LIN {X 70.467,Y 80.092,Z 59.000,A 180.000,B 0.000,C 180.000} C_DIS
LIN {X 70.403,Y 79.913,Z 59.000,A 180.000,B 0.000,C 180.000} C_DIS
LIN {X 70.344,Y 79.735,Z 59.000,A 180.000,B 0.000,C 180.000} C_DIS
LIN {X 70.240,Y 79.377,Z 59.000,A 180.000,B 0.000,C 180.000} C_DIS
LIN {X 70.200,Y 79.198,Z 59.000,A 180.000,B 0.000,C 180.000} C_DIS
LIN {X 70.160,Y 79.020,Z 59.000,A 180.000,B 0.000,C 180.000} C_DIS
LIN {X 70.124,Y 78.841,Z 59.000,A 180.000,B 0.000,C 180.000} C_DIS
LIN {X 70.067,Y 78.483,Z 59.000,A 180.000,B 0.000,C 180.000} C_DIS
LIN {X 70.048,Y 78.304,Z 59.000,A 180.000,B 0.000,C 180.000} C_DIS
LIN {X 70.031,Y 78.126,Z 59.000,A 180.000,B 0.000,C 180.000} C_DIS
LIN {X 70.015,Y 77.947,Z 59.000,A 180.000,B 0.000,C 180.000} C_DIS
LIN {X 70.004,Y 77.589,Z 59.000,A 180.000,B 0.000,C 180.000} C_DIS
LIN {X 70.004,Y 77.411,Z 59.000,A 180.000,B 0.000,C 180.000} C_DIS
LIN {X 70.015,Y 77.053,Z 59.000,A 180.000,B 0.000,C 180.000} C_DIS
LIN {X 70.031,Y 76.874,Z 59.000,A 180.000,B 0.000,C 180.000} C_DIS
LIN {X 70.048,Y 76.696,Z 59.000,A 180.000,B 0.000,C 180.000} C_DIS
LIN {X 70.067,Y 76.517,Z 59.000,A 180.000,B 0.000,C 180.000} C_DIS
LIN {X 70.124,Y 76.159,Z 59.000,A 180.000,B 0.000,C 180.000} C_DIS
LIN {X 70.160,Y 75.980,Z 59.000,A 180.000,B 0.000,C 180.000} C_DIS
LIN {X 70.200,Y 75.802,Z 59.000,A 180.000,B 0.000,C 180.000} C_DIS
LIN {X 70.240,Y 75.623,Z 59.000,A 180.000,B 0.000,C 180.000} C_DIS
LIN {X 70.344,Y 75.265,Z 59.000,A 180.000,B 0.000,C 180.000} C_DIS
LIN {X 70.403,Y 75.087,Z 59.000,A 180.000,B 0.000,C 180.000} C_DIS
LIN {X 70.467,Y 74.908,Z 59.000,A 180.000,B 0.000,C 180.000} C_DIS
LIN {X 70.501,Y 74.814,Z 59.000,A 180.000,B 0.000,C 180.000} C_DIS
LIN {X 70.532,Y 74.729,Z 59.000,A 180.000,B 0.000,C 180.000} C_DIS
LIN {X 70.687,Y 74.372,Z 59.000,A 180.000,B 0.000,C 180.000} C_DIS
LIN {X 70.773,Y 74.193,Z 59.000,A 180.000,B 0.000,C 180.000} C_DIS
LIN {X 70.864,Y 74.014,Z 59.000,A 180.000,B 0.000,C 180.000} C_DIS
LIN {X 70.960,Y 73.835,Z 59.000,A 180.000,B 0.000,C 180.000} C_DIS
LIN {X 71.154,Y 73.507,Z 59.000,A 180.000,B 0.000,C 180.000} C_DIS
LIN {X 71.171,Y 73.478,Z 59.000,A 180.000,B 0.000,C 180.000} C_DIS
LIN {X 71.414,Y 73.120,Z 59.000,A 180.000,B 0.000,C 180.000} C_DIS
LIN {X 71.511,Y 72.992,Z 59.000,A 180.000,B 0.000,C 180.000} C_DIS
LIN {X 71.690,Y 72.762,Z 59.000,A 180.000,B 0.000,C 180.000} C_DIS
LIN {X 71.842,Y 72.584,Z 59.000,A 180.000,B 0.000,C 180.000} C_DIS
LIN {X 72.000,Y 72.405,Z 59.000,A 180.000,B 0.000,C 180.000} C_DIS
LIN {X 72.048,Y 72.353,Z 59.000,A 180.000,B 0.000,C 180.000} C_DIS
LIN {X 72.353,Y 72.048,Z 59.000,A 180.000,B 0.000,C 180.000} C_DIS
LIN {X 72.405,Y 72.000,Z 59.000,A 180.000,B 0.000,C 180.000} C_DIS
LIN {X 72.584,Y 71.842,Z 59.000,A 180.000,B 0.000,C 180.000} C_DIS
LIN {X 72.762,Y 71.690,Z 59.000,A 180.000,B 0.000,C 180.000} C_DIS
LIN {X 72.992,Y 71.511,Z 59.000,A 180.000,B 0.000,C 180.000} C_DIS
LIN {X 73.120,Y 71.414,Z 59.000,A 180.000,B 0.000,C 180.000} C_DIS
LIN {X 73.478,Y 71.171,Z 59.000,A 180.000,B 0.000,C 180.000} C_DIS
LIN {X 73.507,Y 71.154,Z 59.000,A 180.000,B 0.000,C 180.000} C_DIS
LIN {X 73.835,Y 70.960,Z 59.000,A 180.000,B 0.000,C 180.000} C_DIS
LIN {X 74.014,Y 70.864,Z 59.000,A 180.000,B 0.000,C 180.000} C_DIS
LIN {X 74.193,Y 70.773,Z 59.000,A 180.000,B 0.000,C 180.000} C_DIS
LIN {X 74.372,Y 70.687,Z 59.000,A 180.000,B 0.000,C 180.000} C_DIS
LIN {X 74.729,Y 70.532,Z 59.000,A 180.000,B 0.000,C 180.000} C_DIS
LIN {X 74.908,Y 70.467,Z 59.000,A 180.000,B 0.000,C 180.000} C_DIS
LIN {X 75.087,Y 70.403,Z 59.000,A 180.000,B 0.000,C 180.000} C_DIS
LIN {X 75.265,Y 70.344,Z 59.000,A 180.000,B 0.000,C 180.000} C_DIS
LIN {X 75.623,Y 70.240,Z 59.000,A 180.000,B 0.000,C 180.000} C_DIS
LIN {X 75.802,Y 70.200,Z 59.000,A 180.000,B 0.000,C 180.000} C_DIS
LIN {X 75.980,Y 70.160,Z 59.000,A 180.000,B 0.000,C 180.000} C_DIS
LIN {X 76.159,Y 70.124,Z 59.000,A 180.000,B 0.000,C 180.000} C_DIS
LIN {X 76.517,Y 70.067,Z 59.000,A 180.000,B 0.000,C 180.000} C_DIS
LIN {X 76.696,Y 70.048,Z 59.000,A 180.000,B 0.000,C 180.000} C_DIS
LIN {X 76.874,Y 70.031,Z 59.000,A 180.000,B 0.000,C 180.000} C_DIS
LIN {X 77.053,Y 70.015,Z 59.000,A 180.000,B 0.000,C 180.000} C_DIS
LIN {X 77.411,Y 70.004,Z 59.000,A 180.000,B 0.000,C 180.000} C_DIS
LIN {X 77.589,Y 70.004,Z 59.000,A 180.000,B 0.000,C 180.000} C_DIS
LIN {X 77.947,Y 70.015,Z 59.000,A 180.000,B 0.000,C 180.000} C_DIS
LIN {X 78.126,Y 70.031,Z 59.000,A 180.000,B 0.000,C 180.000} C_DIS
LIN {X 78.304,Y 70.048,Z 59.000,A 180.000,B 0.000,C 180.000} C_DIS
LIN {X 78.483,Y 70.067,Z 59.000,A 180.000,B 0.000,C 180.000} C_DIS
LIN {X 78.841,Y 70.124,Z 59.000,A 180.000,B 0.000,C 180.000} C_DIS
LIN {X 79.020,Y 70.160,Z 59.000,A 180.000,B 0.000,C 180.000} C_DIS
LIN {X 79.198,Y 70.200,Z 59.000,A 180.000,B 0.000,C 180.000} C_DIS
LIN {X 79.377,Y 70.240,Z 59.000,A 180.000,B 0.000,C 180.000} C_DIS
LIN {X 79.735,Y 70.344,Z 59.000,A 180.000,B 0.000,C 180.000} C_DIS
LIN {X 79.913,Y 70.403,Z 59.000,A 180.000,B 0.000,C 180.000} C_DIS
LIN {X 80.092,Y 70.467,Z 59.000,A 180.000,B 0.000,C 180.000} C_DIS
LIN {X 80.271,Y 70.532,Z 59.000,A 180.000,B 0.000,C 180.000} C_DIS
LIN {X 80.628,Y 70.687,Z 59.000,A 180.000,B 0.000,C 180.000} C_DIS
LIN {X 80.807,Y 70.773,Z 59.000,A 180.000,B 0.000,C 180.000} C_DIS
LIN {X 80.986,Y 70.864,Z 59.000,A 180.000,B 0.000,C 180.000} C_DIS
LIN {X 81.165,Y 70.960,Z 59.000,A 180.000,B 0.000,C 180.000} C_DIS
LIN {X 81.493,Y 71.154,Z 59.000,A 180.000,B 0.000,C 180.000} C_DIS
LIN {X 81.522,Y 71.171,Z 59.000,A 180.000,B 0.000,C 180.000} C_DIS
LIN {X 81.880,Y 71.414,Z 59.000,A 180.000,B 0.000,C 180.000} C_DIS
LIN {X 82.008,Y 71.511,Z 59.000,A 180.000,B 0.000,C 180.000} C_DIS
LIN {X 82.238,Y 71.690,Z 59.000,A 180.000,B 0.000,C 180.000} C_DIS
LIN {X 82.416,Y 71.842,Z 59.000,A 180.000,B 0.000,C 180.000} C_DIS
LIN {X 82.595,Y 72.000,Z 59.000,A 180.000,B 0.000,C 180.000} C_DIS
LIN {X 82.647,Y 72.048,Z 59.000,A 180.000,B 0.000,C 180.000} C_DIS
LIN {X 82.952,Y 72.353,Z 59.000,A 180.000,B 0.000,C 180.000} C_DIS
LIN {X 83.000,Y 72.405,Z 59.000,A 180.000,B 0.000,C 180.000} C_DIS
LIN {X 83.158,Y 72.584,Z 59.000,A 180.000,B 0.000,C 180.000} C_DIS
LIN {X 83.310,Y 72.762,Z 59.000,A 180.000,B 0.000,C 180.000} C_DIS
LIN {X 83.489,Y 72.992,Z 59.000,A 180.000,B 0.000,C 180.000} C_DIS
LIN {X 83.586,Y 73.120,Z 59.000,A 180.000,B 0.000,C 180.000} C_DIS
LIN {X 83.829,Y 73.478,Z 59.000,A 180.000,B 0.000,C 180.000} C_DIS
LIN {X 83.846,Y 73.507,Z 59.000,A 180.000,B 0.000,C 180.000} C_DIS
LIN {X 84.040,Y 73.835,Z 59.000,A 180.000,B 0.000,C 180.000} C_DIS
LIN {X 84.136,Y 74.014,Z 59.000,A 180.000,B 0.000,C 180.000} C_DIS
LIN {X 84.227,Y 74.193,Z 59.000,A 180.000,B 0.000,C 180.000} C_DIS
LIN {X 84.313,Y 74.372,Z 59.000,A 180.000,B 0.000,C 180.000} C_DIS
LIN {X 84.468,Y 74.729,Z 59.000,A 180.000,B 0.000,C 180.000} C_DIS
LIN {X 84.533,Y 74.908,Z 59.000,A 180.000,B 0.000,C 180.000} C_DIS
LIN {X 84.597,Y 75.087,Z 59.000,A 180.000,B 0.000,C 180.000} C_DIS
LIN {X 84.656,Y 75.265,Z 59.000,A 180.000,B 0.000,C 180.000} C_DIS
LIN {X 84.760,Y 75.623,Z 59.000,A 180.000,B 0.000,C 180.000} C_DIS
LIN {X 84.800,Y 75.802,Z 59.000,A 180.000,B 0.000,C 180.000} C_DIS
LIN {X 84.840,Y 75.980,Z 59.000,A 180.000,B 0.000,C 180.000} C_DIS
LIN {X 84.876,Y 76.159,Z 59.000,A 180.000,B 0.000,C 180.000} C_DIS
LIN {X 84.933,Y 76.517,Z 59.000,A 180.000,B 0.000,C 180.000} C_DIS
LIN {X 84.952,Y 76.696,Z 59.000,A 180.000,B 0.000,C 180.000} C_DIS
LIN {X 84.969,Y 76.874,Z 59.000,A 180.000,B 0.000,C 180.000} C_DIS
LIN {X 84.985,Y 77.053,Z 59.000,A 180.000,B 0.000,C 180.000} C_DIS
LIN {X 84.996,Y 77.411,Z 59.000,A 180.000,B 0.000,C 180.000} C_DIS
LIN {X 84.996,Y 77.589,Z 59.000,A 180.000,B 0.000,C 180.000} C_DIS
LIN {X 84.985,Y 77.947,Z 59.000,A 180.000,B 0.000,C 180.000} C_DIS
LIN {X 84.969,Y 78.126,Z 59.000,A 180.000,B 0.000,C 180.000} C_DIS
LIN {X 84.952,Y 78.304,Z 59.000,A 180.000,B 0.000,C 180.000} C_DIS
LIN {X 84.933,Y 78.483,Z 59.000,A 180.000,B 0.000,C 180.000} C_DIS
LIN {X 84.876,Y 78.841,Z 59.000,A 180.000,B 0.000,C 180.000} C_DIS
LIN {X 84.840,Y 79.020,Z 59.000,A 180.000,B 0.000,C 180.000} C_DIS
LIN {X 84.800,Y 79.198,Z 59.000,A 180.000,B 0.000,C 180.000} C_DIS
LIN {X 84.760,Y 79.377,Z 59.000,A 180.000,B 0.000,C 180.000} C_DIS
LIN {X 84.656,Y 79.735,Z 59.000,A 180.000,B 0.000,C 180.000} C_DIS
LIN {X 84.597,Y 79.913,Z 59.000,A 180.000,B 0.000,C 180.000} C_DIS
LIN {X 84.533,Y 80.092,Z 59.000,A 180.000,B 0.000,C 180.000} C_DIS
LIN {X 84.468,Y 80.271,Z 59.000,A 180.000,B 0.000,C 180.000} C_DIS
LIN {X 84.313,Y 80.628,Z 59.000,A 180.000,B 0.000,C 180.000} C_DIS
LIN {X 84.227,Y 80.807,Z 59.000,A 180.000,B 0.000,C 180.000} C_DIS
LIN {X 84.136,Y 80.986,Z 59.000,A 180.000,B 0.000,C 180.000} C_DIS
LIN {X 84.040,Y 81.165,Z 59.000,A 180.000,B 0.000,C 180.000} C_DIS
LIN {X 83.846,Y 81.493,Z 59.000,A 180.000,B 0.000,C 180.000} C_DIS
LIN {X 83.829,Y 81.522,Z 59.000,A 180.000,B 0.000,C 180.000} C_DIS
LIN {X 83.586,Y 81.880,Z 59.000,A 180.000,B 0.000,C 180.000} C_DIS
LIN {X 83.489,Y 82.008,Z 59.000,A 180.000,B 0.000,C 180.000} C_DIS
LIN {X 83.310,Y 82.238,Z 59.000,A 180.000,B 0.000,C 180.000} C_DIS
LIN {X 83.158,Y 82.416,Z 59.000,A 180.000,B 0.000,C 180.000} C_DIS
LIN {X 83.000,Y 82.595,Z 59.000,A 180.000,B 0.000,C 180.000} C_DIS
LIN {X 82.952,Y 82.647,Z 59.000,A 180.000,B 0.000,C 180.000} C_DIS
LIN {X 82.647,Y 82.952,Z 59.000,A 180.000,B 0.000,C 180.000} C_DIS
LIN {X 82.595,Y 83.000,Z 59.000,A 180.000,B 0.000,C 180.000} C_DIS
LIN {X 82.416,Y 83.158,Z 59.000,A 180.000,B 0.000,C 180.000} C_DIS
LIN {X 82.238,Y 83.310,Z 59.000,A 180.000,B 0.000,C 180.000} C_DIS
LIN {X 82.008,Y 83.489,Z 59.000,A 180.000,B 0.000,C 180.000} C_DIS
LIN {X 81.880,Y 83.586,Z 59.000,A 180.000,B 0.000,C 180.000} C_DIS
LIN {X 81.522,Y 83.829,Z 59.000,A 180.000,B 0.000,C 180.000} C_DIS
LIN {X 81.493,Y 83.846,Z 59.000,A 180.000,B 0.000,C 180.000} C_DIS
LIN {X 81.165,Y 84.040,Z 59.000,A 180.000,B 0.000,C 180.000} C_DIS
LIN {X 80.986,Y 84.136,Z 59.000,A 180.000,B 0.000,C 180.000} C_DIS
LIN {X 80.807,Y 84.227,Z 59.000,A 180.000,B 0.000,C 180.000} C_DIS
LIN {X 80.628,Y 84.313,Z 59.000,A 180.000,B 0.000,C 180.000} C_DIS
LIN {X 80.271,Y 84.468,Z 59.000,A 180.000,B 0.000,C 180.000} C_DIS
LIN {X 80.092,Y 84.533,Z 59.000,A 180.000,B 0.000,C 180.000} C_DIS
LIN {X 79.913,Y 84.597,Z 59.000,A 180.000,B 0.000,C 180.000} C_DIS
LIN {X 79.735,Y 84.656,Z 59.000,A 180.000,B 0.000,C 180.000} C_DIS
LIN {X 79.377,Y 84.760,Z 59.000,A 180.000,B 0.000,C 180.000} C_DIS
LIN {X 79.198,Y 84.800,Z 59.000,A 180.000,B 0.000,C 180.000} C_DIS
LIN {X 79.020,Y 84.840,Z 59.000,A 180.000,B 0.000,C 180.000} C_DIS
LIN {X 78.841,Y 84.876,Z 59.000,A 180.000,B 0.000,C 180.000} C_DIS
LIN {X 78.483,Y 84.933,Z 59.000,A 180.000,B 0.000,C 180.000} C_DIS
LIN {X 78.304,Y 84.952,Z 59.000,A 180.000,B 0.000,C 180.000} C_DIS
LIN {X 78.126,Y 84.969,Z 59.000,A 180.000,B 0.000,C 180.000} C_DIS
LIN {X 77.947,Y 84.985,Z 59.000,A 180.000,B 0.000,C 180.000} C_DIS
LIN {X 77.589,Y 84.996,Z 59.000,A 180.000,B 0.000,C 180.000} C_DIS
LIN {X 77.411,Y 84.996,Z 59.000,A 180.000,B 0.000,C 180.000} C_DIS
LIN {X 77.053,Y 84.985,Z 59.000,A 180.000,B 0.000,C 180.000} C_DIS
LIN {X 76.874,Y 84.969,Z 59.000,A 180.000,B 0.000,C 180.000} C_DIS
LIN {X 76.696,Y 84.952,Z 59.000,A 180.000,B 0.000,C 180.000} C_DIS
LIN {X 76.517,Y 84.933,Z 59.000,A 180.000,B 0.000,C 180.000} C_DIS
LIN {X 76.159,Y 84.876,Z 59.000,A 180.000,B 0.000,C 180.000} C_DIS
LIN {X 75.980,Y 84.840,Z 59.000,A 180.000,B 0.000,C 180.000} C_DIS
LIN {X 75.802,Y 84.800,Z 59.000,A 180.000,B 0.000,C 180.000} C_DIS
LIN {X 75.623,Y 84.760,Z 59.000,A 180.000,B 0.000,C 180.000} C_DIS
LIN {X 75.265,Y 84.656,Z 59.000,A 180.000,B 0.000,C 180.000} C_DIS
LIN {X 75.087,Y 84.597,Z 59.000,A 180.000,B 0.000,C 180.000} C_DIS
LIN {X 74.908,Y 84.533,Z 59.000,A 180.000,B 0.000,C 180.000} C_DIS
LIN {X 74.729,Y 84.468,Z 59.000,A 180.000,B 0.000,C 180.000} C_DIS
LIN {X 74.372,Y 84.313,Z 59.000,A 180.000,B 0.000,C 180.000} C_DIS
LIN {X 74.193,Y 84.227,Z 59.000,A 180.000,B 0.000,C 180.000} C_DIS
LIN {X 74.014,Y 84.136,Z 59.000,A 180.000,B 0.000,C 180.000} C_DIS
LIN {X 73.835,Y 84.040,Z 59.000,A 180.000,B 0.000,C 180.000} C_DIS
LIN {X 73.507,Y 83.846,Z 59.000,A 180.000,B 0.000,C 180.000} C_DIS
LIN {X 73.478,Y 83.829,Z 59.000,A 180.000,B 0.000,C 180.000} C_DIS
LIN {X 73.260,Y 83.681,Z 59.000,A 180.000,B 0.000,C 180.000} C_DIS
; Link Move Starts
LIN {X 73.004,Y 83.498,Z 59.000,A 180.000,B 0.000,C 180.000} C_DIS
LIN {X 72.755,Y 83.305,Z 58.999,A 180.000,B 0.000,C 180.000} C_DIS
LIN {X 72.517,Y 83.099,Z 58.998,A 180.000,B 0.000,C 180.000} C_DIS
LIN {X 72.286,Y 82.885,Z 58.996,A 180.000,B 0.000,C 180.000} C_DIS
LIN {X 72.063,Y 82.663,Z 58.994,A 180.000,B 0.000,C 180.000} C_DIS
LIN {X 71.853,Y 82.428,Z 58.991,A 180.000,B 0.000,C 180.000} C_DIS
LIN {X 71.650,Y 82.187,Z 58.988,A 180.000,B 0.000,C 180.000} C_DIS
LIN {X 71.457,Y 81.938,Z 58.985,A 180.000,B 0.000,C 180.000} C_DIS
LIN {X 71.278,Y 81.679,Z 58.981,A 180.000,B 0.000,C 180.000} C_DIS
LIN {X 71.107,Y 81.414,Z 58.977,A 180.000,B 0.000,C 180.000} C_DIS
LIN {X 70.947,Y 81.143,Z 58.972,A 180.000,B 0.000,C 180.000} C_DIS
LIN {X 70.873,Y 81.004,Z 58.969,A 180.000,B 0.000,C 180.000} C_DIS
LIN {X 70.802,Y 80.864,Z 58.967,A 180.000,B 0.000,C 180.000} C_DIS
LIN {X 70.730,Y 80.723,Z 58.964,A 180.000,B 0.000,C 180.000} C_DIS
LIN {X 70.666,Y 80.579,Z 58.961,A 180.000,B 0.000,C 180.000} C_DIS
LIN {X 70.603,Y 80.435,Z 58.959,A 180.000,B 0.000,C 180.000} C_DIS
LIN {X 70.541,Y 80.290,Z 58.956,A 180.000,B 0.000,C 180.000} C_DIS
LIN {X 70.485,Y 80.143,Z 58.952,A 180.000,B 0.000,C 180.000} C_DIS
LIN {X 70.432,Y 79.995,Z 58.949,A 180.000,B 0.000,C 180.000} C_DIS
LIN {X 70.379,Y 79.847,Z 58.946,A 180.000,B 0.000,C 180.000} C_DIS
LIN {X 70.333,Y 79.696,Z 58.943,A 180.000,B 0.000,C 180.000} C_DIS
LIN {X 70.289,Y 79.545,Z 58.939,A 180.000,B 0.000,C 180.000} C_DIS
LIN {X 70.245,Y 79.393,Z 58.936,A 180.000,B 0.000,C 180.000} C_DIS
LIN {X 70.209,Y 79.240,Z 58.932,A 180.000,B 0.000,C 180.000} C_DIS
LIN {X 70.175,Y 79.086,Z 58.928,A 180.000,B 0.000,C 180.000} C_DIS
LIN {X 70.140,Y 78.933,Z 58.925,A 180.000,B 0.000,C 180.000} C_DIS
LIN {X 70.114,Y 78.777,Z 58.921,A 180.000,B 0.000,C 180.000} C_DIS
LIN {X 70.089,Y 78.622,Z 58.917,A 180.000,B 0.000,C 180.000} C_DIS
LIN {X 70.065,Y 78.466,Z 58.913,A 180.000,B 0.000,C 180.000} C_DIS
LIN {X 70.048,Y 78.310,Z 58.909,A 180.000,B 0.000,C 180.000} C_DIS
LIN {X 70.033,Y 78.153,Z 58.905,A 180.000,B 0.000,C 180.000} C_DIS
LIN {X 70.018,Y 77.996,Z 58.900,A 180.000,B 0.000,C 180.000} C_DIS
LIN {X 70.012,Y 77.839,Z 58.896,A 180.000,B 0.000,C 180.000} C_DIS
LIN {X 70.007,Y 77.681,Z 58.892,A 180.000,B 0.000,C 180.000} C_DIS
LIN {X 70.002,Y 77.524,Z 58.887,A 180.000,B 0.000,C 180.000} C_DIS
LIN {X 70.005,Y 77.366,Z 58.883,A 180.000,B 0.000,C 180.000} C_DIS
LIN {X 70.010,Y 77.209,Z 58.878,A 180.000,B 0.000,C 180.000} C_DIS
LIN {X 70.015,Y 77.051,Z 58.873,A 180.000,B 0.000,C 180.000} C_DIS
LIN {X 70.029,Y 76.894,Z 58.869,A 180.000,B 0.000,C 180.000} C_DIS
LIN {X 70.044,Y 76.738,Z 58.864,A 180.000,B 0.000,C 180.000} C_DIS
LIN {X 70.058,Y 76.581,Z 58.859,A 180.000,B 0.000,C 180.000} C_DIS
LIN {X 70.082,Y 76.425,Z 58.854,A 180.000,B 0.000,C 180.000} C_DIS
LIN {X 70.094,Y 76.347,Z 58.851,A 180.000,B 0.000,C 180.000} C_DIS
LIN {X 70.106,Y 76.270,Z 58.849,A 180.000,B 0.000,C 180.000} C_DIS
LIN {X 70.119,Y 76.192,Z 58.846,A 180.000,B 0.000,C 180.000} C_DIS
LIN {X 70.131,Y 76.114,Z 58.844,A 180.000,B 0.000,C 180.000} C_DIS
LIN {X 70.147,Y 76.037,Z 58.841,A 180.000,B 0.000,C 180.000} C_DIS
LIN {X 70.164,Y 75.960,Z 58.839,A 180.000,B 0.000,C 180.000} C_DIS
LIN {X 70.181,Y 75.883,Z 58.836,A 180.000,B 0.000,C 180.000} C_DIS
LIN {X 70.216,Y 75.729,Z 58.831,A 180.000,B 0.000,C 180.000} C_DIS
LIN {X 70.233,Y 75.653,Z 58.828,A 180.000,B 0.000,C 180.000} C_DIS
LIN {X 70.254,Y 75.577,Z 58.825,A 180.000,B 0.000,C 180.000} C_DIS
LIN {X 70.298,Y 75.425,Z 58.820,A 180.000,B 0.000,C 180.000} C_DIS
LIN {X 70.342,Y 75.274,Z 58.815,A 180.000,B 0.000,C 180.000} C_DIS
LIN {X 70.364,Y 75.198,Z 58.812,A 180.000,B 0.000,C 180.000} C_DIS
LIN {X 70.389,Y 75.124,Z 58.809,A 180.000,B 0.000,C 180.000} C_DIS
LIN {X 70.416,Y 75.050,Z 58.806,A 180.000,B 0.000,C 180.000} C_DIS
LIN {X 70.469,Y 74.902,Z 58.801,A 180.000,B 0.000,C 180.000} C_DIS
LIN {X 70.523,Y 74.754,Z 58.796,A 180.000,B 0.000,C 180.000} C_DIS
LIN {X 70.553,Y 74.681,Z 58.793,A 180.000,B 0.000,C 180.000} C_DIS
LIN {X 70.616,Y 74.536,Z 58.787,A 180.000,B 0.000,C 180.000} C_DIS
LIN {X 70.647,Y 74.464,Z 58.785,A 180.000,B 0.000,C 180.000} C_DIS
LIN {X 70.710,Y 74.320,Z 58.779,A 180.000,B 0.000,C 180.000} C_DIS
LIN {X 70.745,Y 74.249,Z 58.776,A 180.000,B 0.000,C 180.000} C_DIS
LIN {X 70.780,Y 74.179,Z 58.774,A 180.000,B 0.000,C 180.000} C_DIS
LIN {X 70.852,Y 74.038,Z 58.768,A 180.000,B 0.000,C 180.000} C_DIS
LIN {X 70.923,Y 73.898,Z 58.763,A 180.000,B 0.000,C 180.000} C_DIS
LIN {X 70.963,Y 73.830,Z 58.760,A 180.000,B 0.000,C 180.000} C_DIS
LIN {X 71.043,Y 73.694,Z 58.754,A 180.000,B 0.000,C 180.000} C_DIS
LIN {X 71.083,Y 73.627,Z 58.752,A 180.000,B 0.000,C 180.000} C_DIS
LIN {X 71.163,Y 73.491,Z 58.746,A 180.000,B 0.000,C 180.000} C_DIS
LIN {X 71.207,Y 73.425,Z 58.743,A 180.000,B 0.000,C 180.000} C_DIS
LIN {X 71.251,Y 73.360,Z 58.741,A 180.000,B 0.000,C 180.000} C_DIS
LIN {X 71.340,Y 73.230,Z 58.735,A 180.000,B 0.000,C 180.000} C_DIS
LIN {X 71.428,Y 73.100,Z 58.730,A 180.000,B 0.000,C 180.000} C_DIS
LIN {X 71.476,Y 73.037,Z 58.727,A 180.000,B 0.000,C 180.000} C_DIS
LIN {X 71.573,Y 72.913,Z 58.721,A 180.000,B 0.000,C 180.000} C_DIS
LIN {X 71.621,Y 72.851,Z 58.719,A 180.000,B 0.000,C 180.000} C_DIS
LIN {X 71.717,Y 72.726,Z 58.713,A 180.000,B 0.000,C 180.000} C_DIS
LIN {X 71.769,Y 72.667,Z 58.710,A 180.000,B 0.000,C 180.000} C_DIS
LIN {X 71.821,Y 72.608,Z 58.708,A 180.000,B 0.000,C 180.000} C_DIS
LIN {X 71.925,Y 72.489,Z 58.702,A 180.000,B 0.000,C 180.000} C_DIS
LIN {X 72.030,Y 72.371,Z 58.697,A 180.000,B 0.000,C 180.000} C_DIS
LIN {X 72.085,Y 72.315,Z 58.694,A 180.000,B 0.000,C 180.000} C_DIS
LIN {X 72.196,Y 72.204,Z 58.688,A 180.000,B 0.000,C 180.000} C_DIS
LIN {X 72.252,Y 72.148,Z 58.686,A 180.000,B 0.000,C 180.000} C_DIS
LIN {X 72.363,Y 72.037,Z 58.680,A 180.000,B 0.000,C 180.000} C_DIS
LIN {X 72.422,Y 71.985,Z 58.677,A 180.000,B 0.000,C 180.000} C_DIS
LIN {X 72.541,Y 71.880,Z 58.672,A 180.000,B 0.000,C 180.000} C_DIS
LIN {X 72.659,Y 71.776,Z 58.666,A 180.000,B 0.000,C 180.000} C_DIS
LIN {X 72.718,Y 71.724,Z 58.664,A 180.000,B 0.000,C 180.000} C_DIS
LIN {X 72.780,Y 71.676,Z 58.661,A 180.000,B 0.000,C 180.000} C_DIS
LIN {X 73.091,Y 71.434,Z 58.647,A 180.000,B 0.000,C 180.000} C_DIS
LIN {X 73.156,Y 71.390,Z 58.644,A 180.000,B 0.000,C 180.000} C_DIS
LIN {X 73.286,Y 71.301,Z 58.639,A 180.000,B 0.000,C 180.000} C_DIS
LIN {X 73.482,Y 71.169,Z 58.631,A 180.000,B 0.000,C 180.000} C_DIS
LIN {X 73.617,Y 71.089,Z 58.625,A 180.000,B 0.000,C 180.000} C_DIS
LIN {X 73.821,Y 70.968,Z 58.617,A 180.000,B 0.000,C 180.000} C_DIS
LIN {X 73.889,Y 70.928,Z 58.614,A 180.000,B 0.000,C 180.000} C_DIS
LIN {X 74.239,Y 70.749,Z 58.600,A 180.000,B 0.000,C 180.000} C_DIS
LIN {X 74.310,Y 70.714,Z 58.598,A 180.000,B 0.000,C 180.000} C_DIS
LIN {X 74.527,Y 70.620,Z 58.589,A 180.000,B 0.000,C 180.000} C_DIS
LIN {X 74.671,Y 70.557,Z 58.584,A 180.000,B 0.000,C 180.000} C_DIS
LIN {X 74.743,Y 70.526,Z 58.581,A 180.000,B 0.000,C 180.000} C_DIS
LIN {X 75.114,Y 70.393,Z 58.567,A 180.000,B 0.000,C 180.000} C_DIS
LIN {X 75.188,Y 70.367,Z 58.565,A 180.000,B 0.000,C 180.000} C_DIS
LIN {X 75.566,Y 70.257,Z 58.551,A 180.000,B 0.000,C 180.000} C_DIS
LIN {X 75.642,Y 70.235,Z 58.548,A 180.000,B 0.000,C 180.000} C_DIS
LIN {X 76.026,Y 70.149,Z 58.534,A 180.000,B 0.000,C 180.000} C_DIS
LIN {X 76.103,Y 70.133,Z 58.532,A 180.000,B 0.000,C 180.000} C_DIS
LIN {X 76.492,Y 70.071,Z 58.518,A 180.000,B 0.000,C 180.000} C_DIS
LIN {X 76.570,Y 70.059,Z 58.515,A 180.000,B 0.000,C 180.000} C_DIS
LIN {X 76.962,Y 70.022,Z 58.501,A 180.000,B 0.000,C 180.000} C_DIS
LIN {X 77.041,Y 70.016,Z 58.499,A 180.000,B 0.000,C 180.000} C_DIS
LIN {X 77.434,Y 70.003,Z 58.485,A 180.000,B 0.000,C 180.000} C_DIS
LIN {X 77.513,Y 70.002,Z 58.482,A 180.000,B 0.000,C 180.000} C_DIS
LIN {X 77.907,Y 70.014,Z 58.468,A 180.000,B 0.000,C 180.000} C_DIS
LIN {X 77.985,Y 70.017,Z 58.466,A 180.000,B 0.000,C 180.000} C_DIS
LIN {X 78.377,Y 70.054,Z 58.452,A 180.000,B 0.000,C 180.000} C_DIS
LIN {X 78.456,Y 70.063,Z 58.449,A 180.000,B 0.000,C 180.000} C_DIS
LIN {X 78.845,Y 70.124,Z 58.435,A 180.000,B 0.000,C 180.000} C_DIS
LIN {X 78.922,Y 70.138,Z 58.433,A 180.000,B 0.000,C 180.000} C_DIS
LIN {X 79.307,Y 70.224,Z 58.419,A 180.000,B 0.000,C 180.000} C_DIS
LIN {X 79.383,Y 70.242,Z 58.416,A 180.000,B 0.000,C 180.000} C_DIS
LIN {X 79.761,Y 70.352,Z 58.402,A 180.000,B 0.000,C 180.000} C_DIS
LIN {X 79.836,Y 70.375,Z 58.400,A 180.000,B 0.000,C 180.000} C_DIS
LIN {X 80.059,Y 70.455,Z 58.391,A 180.000,B 0.000,C 180.000} C_DIS
LIN {X 80.207,Y 70.509,Z 58.386,A 180.000,B 0.000,C 180.000} C_DIS
LIN {X 80.281,Y 70.537,Z 58.383,A 180.000,B 0.000,C 180.000} C_DIS
LIN {X 80.642,Y 70.693,Z 58.369,A 180.000,B 0.000,C 180.000} C_DIS
LIN {X 80.714,Y 70.726,Z 58.367,A 180.000,B 0.000,C 180.000} C_DIS
LIN {X 80.924,Y 70.833,Z 58.358,A 180.000,B 0.000,C 180.000} C_DIS
LIN {X 81.065,Y 70.904,Z 58.353,A 180.000,B 0.000,C 180.000} C_DIS
LIN {X 81.134,Y 70.941,Z 58.350,A 180.000,B 0.000,C 180.000} C_DIS
LIN {X 81.473,Y 71.142,Z 58.336,A 180.000,B 0.000,C 180.000} C_DIS
LIN {X 81.540,Y 71.183,Z 58.334,A 180.000,B 0.000,C 180.000} C_DIS
LIN {X 81.670,Y 71.272,Z 58.328,A 180.000,B 0.000,C 180.000} C_DIS
LIN {X 81.865,Y 71.405,Z 58.320,A 180.000,B 0.000,C 180.000} C_DIS
LIN {X 81.930,Y 71.450,Z 58.317,A 180.000,B 0.000,C 180.000} C_DIS
LIN {X 82.241,Y 71.692,Z 58.303,A 180.000,B 0.000,C 180.000} C_DIS
LIN {X 82.302,Y 71.741,Z 58.301,A 180.000,B 0.000,C 180.000} C_DIS
LIN {X 82.420,Y 71.846,Z 58.295,A 180.000,B 0.000,C 180.000} C_DIS
LIN {X 82.597,Y 72.002,Z 58.287,A 180.000,B 0.000,C 180.000} C_DIS
LIN {X 82.655,Y 72.055,Z 58.284,A 180.000,B 0.000,C 180.000} C_DIS
LIN {X 82.822,Y 72.222,Z 58.276,A 180.000,B 0.000,C 180.000} C_DIS
LIN {X 82.933,Y 72.334,Z 58.270,A 180.000,B 0.000,C 180.000} C_DIS
LIN {X 82.988,Y 72.391,Z 58.268,A 180.000,B 0.000,C 180.000} C_DIS
LIN {X 83.092,Y 72.509,Z 58.262,A 180.000,B 0.000,C 180.000} C_DIS
LIN {X 83.248,Y 72.686,Z 58.254,A 180.000,B 0.000,C 180.000} C_DIS
LIN {X 83.299,Y 72.747,Z 58.251,A 180.000,B 0.000,C 180.000} C_DIS
LIN {X 83.443,Y 72.933,Z 58.243,A 180.000,B 0.000,C 180.000} C_DIS
LIN {X 83.540,Y 73.058,Z 58.237,A 180.000,B 0.000,C 180.000} C_DIS
LIN {X 83.586,Y 73.121,Z 58.235,A 180.000,B 0.000,C 180.000} C_DIS
LIN {X 83.675,Y 73.252,Z 58.229,A 180.000,B 0.000,C 180.000} C_DIS
LIN {X 83.808,Y 73.447,Z 58.221,A 180.000,B 0.000,C 180.000} C_DIS
LIN {X 83.850,Y 73.513,Z 58.218,A 180.000,B 0.000,C 180.000} C_DIS
LIN {X 83.970,Y 73.717,Z 58.210,A 180.000,B 0.000,C 180.000} C_DIS
LIN {X 84.050,Y 73.852,Z 58.204,A 180.000,B 0.000,C 180.000} C_DIS
LIN {X 84.088,Y 73.921,Z 58.202,A 180.000,B 0.000,C 180.000} C_DIS
LIN {X 84.160,Y 74.062,Z 58.196,A 180.000,B 0.000,C 180.000} C_DIS
LIN {X 84.232,Y 74.202,Z 58.191,A 180.000,B 0.000,C 180.000} C_DIS
LIN {X 84.267,Y 74.272,Z 58.188,A 180.000,B 0.000,C 180.000} C_DIS
LIN {X 84.301,Y 74.343,Z 58.185,A 180.000,B 0.000,C 180.000} C_DIS
LIN {X 84.363,Y 74.488,Z 58.180,A 180.000,B 0.000,C 180.000} C_DIS
LIN {X 84.426,Y 74.633,Z 58.174,A 180.000,B 0.000,C 180.000} C_DIS
LIN {X 84.457,Y 74.705,Z 58.172,A 180.000,B 0.000,C 180.000} C_DIS
LIN {X 84.486,Y 74.778,Z 58.169,A 180.000,B 0.000,C 180.000} C_DIS
LIN {X 84.539,Y 74.926,Z 58.164,A 180.000,B 0.000,C 180.000} C_DIS
LIN {X 84.566,Y 75.000,Z 58.161,A 180.000,B 0.000,C 180.000} C_DIS
LIN {X 84.593,Y 75.074,Z 58.159,A 180.000,B 0.000,C 180.000} C_DIS
LIN {X 84.619,Y 75.149,Z 58.156,A 180.000,B 0.000,C 180.000} C_DIS
LIN {X 84.644,Y 75.224,Z 58.154,A 180.000,B 0.000,C 180.000} C_DIS
LIN {X 84.666,Y 75.299,Z 58.151,A 180.000,B 0.000,C 180.000} C_DIS
LIN {X 84.688,Y 75.375,Z 58.149,A 180.000,B 0.000,C 180.000} C_DIS
LIN {X 84.731,Y 75.526,Z 58.144,A 180.000,B 0.000,C 180.000} C_DIS
LIN {X 84.773,Y 75.678,Z 58.139,A 180.000,B 0.000,C 180.000} C_DIS
LIN {X 84.807,Y 75.832,Z 58.134,A 180.000,B 0.000,C 180.000} C_DIS
LIN {X 84.841,Y 75.985,Z 58.129,A 180.000,B 0.000,C 180.000} C_DIS
LIN {X 84.873,Y 76.140,Z 58.124,A 180.000,B 0.000,C 180.000} C_DIS
LIN {X 84.898,Y 76.295,Z 58.120,A 180.000,B 0.000,C 180.000} C_DIS
LIN {X 84.922,Y 76.451,Z 58.115,A 180.000,B 0.000,C 180.000} C_DIS
LIN {X 84.944,Y 76.607,Z 58.111,A 180.000,B 0.000,C 180.000} C_DIS
LIN {X 84.959,Y 76.764,Z 58.106,A 180.000,B 0.000,C 180.000} C_DIS
LIN {X 84.974,Y 76.920,Z 58.102,A 180.000,B 0.000,C 180.000} C_DIS
LIN {X 84.985,Y 77.078,Z 58.097,A 180.000,B 0.000,C 180.000} C_DIS
LIN {X 84.990,Y 77.235,Z 58.093,A 180.000,B 0.000,C 180.000} C_DIS
LIN {X 84.995,Y 77.392,Z 58.089,A 180.000,B 0.000,C 180.000} C_DIS
LIN {X 84.997,Y 77.550,Z 58.085,A 180.000,B 0.000,C 180.000} C_DIS
LIN {X 84.992,Y 77.707,Z 58.081,A 180.000,B 0.000,C 180.000} C_DIS
LIN {X 84.987,Y 77.865,Z 58.077,A 180.000,B 0.000,C 180.000} C_DIS
LIN {X 84.979,Y 78.022,Z 58.073,A 180.000,B 0.000,C 180.000} C_DIS
LIN {X 84.964,Y 78.179,Z 58.070,A 180.000,B 0.000,C 180.000} C_DIS
LIN {X 84.950,Y 78.336,Z 58.066,A 180.000,B 0.000,C 180.000} C_DIS
LIN {X 84.931,Y 78.492,Z 58.062,A 180.000,B 0.000,C 180.000} C_DIS
LIN {X 84.907,Y 78.648,Z 58.059,A 180.000,B 0.000,C 180.000} C_DIS
LIN {X 84.882,Y 78.803,Z 58.056,A 180.000,B 0.000,C 180.000} C_DIS
LIN {X 84.854,Y 78.958,Z 58.052,A 180.000,B 0.000,C 180.000} C_DIS
LIN {X 84.820,Y 79.112,Z 58.049,A 180.000,B 0.000,C 180.000} C_DIS
LIN {X 84.785,Y 79.266,Z 58.046,A 180.000,B 0.000,C 180.000} C_DIS
LIN {X 84.748,Y 79.418,Z 58.043,A 180.000,B 0.000,C 180.000} C_DIS
LIN {X 84.704,Y 79.570,Z 58.040,A 180.000,B 0.000,C 180.000} C_DIS
LIN {X 84.660,Y 79.721,Z 58.037,A 180.000,B 0.000,C 180.000} C_DIS
LIN {X 84.612,Y 79.871,Z 58.034,A 180.000,B 0.000,C 180.000} C_DIS
LIN {X 84.559,Y 80.019,Z 58.032,A 180.000,B 0.000,C 180.000} C_DIS
LIN {X 84.506,Y 80.167,Z 58.029,A 180.000,B 0.000,C 180.000} C_DIS
LIN {X 84.449,Y 80.314,Z 58.027,A 180.000,B 0.000,C 180.000} C_DIS
LIN {X 84.324,Y 80.603,Z 58.022,A 180.000,B 0.000,C 180.000} C_DIS
LIN {X 84.186,Y 80.887,Z 58.018,A 180.000,B 0.000,C 180.000} C_DIS
LIN {X 84.040,Y 81.166,Z 58.014,A 180.000,B 0.000,C 180.000} C_DIS
LIN {X 83.879,Y 81.437,Z 58.011,A 180.000,B 0.000,C 180.000} C_DIS
LIN {X 83.707,Y 81.701,Z 58.008,A 180.000,B 0.000,C 180.000} C_DIS
LIN {X 83.527,Y 81.959,Z 58.005,A 180.000,B 0.000,C 180.000} C_DIS
LIN {X 83.334,Y 82.208,Z 58.003,A 180.000,B 0.000,C 180.000} C_DIS
LIN {X 83.130,Y 82.448,Z 58.002,A 180.000,B 0.000,C 180.000} C_DIS
LIN {X 82.919,Y 82.681,Z 58.001,A 180.000,B 0.000,C 180.000} C_DIS
LIN {X 82.696,Y 82.904,Z 58.000,A 180.000,B 0.000,C 180.000} C_DIS
LIN {X 82.526,Y 83.061,Z 58.000,A 180.000,B 0.000,C 180.000} C_DIS
; Cutting Move Starts
LIN {X 82.416,Y 83.158,Z 58.000,A 180.000,B 0.000,C 180.000} C_DIS
LIN {X 82.238,Y 83.310,Z 58.000,A 180.000,B 0.000,C 180.000} C_DIS
LIN {X 82.008,Y 83.489,Z 58.000,A 180.000,B 0.000,C 180.000} C_DIS
LIN {X 81.880,Y 83.586,Z 58.000,A 180.000,B 0.000,C 180.000} C_DIS
LIN {X 81.522,Y 83.829,Z 58.000,A 180.000,B 0.000,C 180.000} C_DIS
LIN {X 81.493,Y 83.846,Z 58.000,A 180.000,B 0.000,C 180.000} C_DIS
LIN {X 81.165,Y 84.040,Z 58.000,A 180.000,B 0.000,C 180.000} C_DIS
LIN {X 80.986,Y 84.136,Z 58.000,A 180.000,B 0.000,C 180.000} C_DIS
LIN {X 80.807,Y 84.227,Z 58.000,A 180.000,B 0.000,C 180.000} C_DIS
LIN {X 80.628,Y 84.313,Z 58.000,A 180.000,B 0.000,C 180.000} C_DIS
LIN {X 80.271,Y 84.468,Z 58.000,A 180.000,B 0.000,C 180.000} C_DIS
LIN {X 80.092,Y 84.533,Z 58.000,A 180.000,B 0.000,C 180.000} C_DIS
LIN {X 79.913,Y 84.597,Z 58.000,A 180.000,B 0.000,C 180.000} C_DIS
LIN {X 79.735,Y 84.656,Z 58.000,A 180.000,B 0.000,C 180.000} C_DIS
LIN {X 79.377,Y 84.760,Z 58.000,A 180.000,B 0.000,C 180.000} C_DIS
LIN {X 79.198,Y 84.800,Z 58.000,A 180.000,B 0.000,C 180.000} C_DIS
LIN {X 79.020,Y 84.840,Z 58.000,A 180.000,B 0.000,C 180.000} C_DIS
LIN {X 78.841,Y 84.876,Z 58.000,A 180.000,B 0.000,C 180.000} C_DIS
LIN {X 78.483,Y 84.933,Z 58.000,A 180.000,B 0.000,C 180.000} C_DIS
LIN {X 78.304,Y 84.952,Z 58.000,A 180.000,B 0.000,C 180.000} C_DIS
LIN {X 78.126,Y 84.969,Z 58.000,A 180.000,B 0.000,C 180.000} C_DIS
LIN {X 77.947,Y 84.985,Z 58.000,A 180.000,B 0.000,C 180.000} C_DIS
LIN {X 77.589,Y 84.996,Z 58.000,A 180.000,B 0.000,C 180.000} C_DIS
LIN {X 77.411,Y 84.996,Z 58.000,A 180.000,B 0.000,C 180.000} C_DIS
LIN {X 77.053,Y 84.985,Z 58.000,A 180.000,B 0.000,C 180.000} C_DIS
LIN {X 76.874,Y 84.969,Z 58.000,A 180.000,B 0.000,C 180.000} C_DIS
LIN {X 76.696,Y 84.952,Z 58.000,A 180.000,B 0.000,C 180.000} C_DIS
LIN {X 76.517,Y 84.933,Z 58.000,A 180.000,B 0.000,C 180.000} C_DIS
LIN {X 76.159,Y 84.876,Z 58.000,A 180.000,B 0.000,C 180.000} C_DIS
LIN {X 75.980,Y 84.840,Z 58.000,A 180.000,B 0.000,C 180.000} C_DIS
LIN {X 75.802,Y 84.800,Z 58.000,A 180.000,B 0.000,C 180.000} C_DIS
LIN {X 75.623,Y 84.760,Z 58.000,A 180.000,B 0.000,C 180.000} C_DIS
LIN {X 75.265,Y 84.656,Z 58.000,A 180.000,B 0.000,C 180.000} C_DIS
LIN {X 75.087,Y 84.597,Z 58.000,A 180.000,B 0.000,C 180.000} C_DIS
LIN {X 74.908,Y 84.533,Z 58.000,A 180.000,B 0.000,C 180.000} C_DIS
LIN {X 74.729,Y 84.468,Z 58.000,A 180.000,B 0.000,C 180.000} C_DIS
LIN {X 74.372,Y 84.313,Z 58.000,A 180.000,B 0.000,C 180.000} C_DIS
LIN {X 74.193,Y 84.227,Z 58.000,A 180.000,B 0.000,C 180.000} C_DIS
LIN {X 74.014,Y 84.136,Z 58.000,A 180.000,B 0.000,C 180.000} C_DIS
LIN {X 73.835,Y 84.040,Z 58.000,A 180.000,B 0.000,C 180.000} C_DIS
LIN {X 73.507,Y 83.846,Z 58.000,A 180.000,B 0.000,C 180.000} C_DIS
LIN {X 73.478,Y 83.829,Z 58.000,A 180.000,B 0.000,C 180.000} C_DIS
LIN {X 73.260,Y 83.681,Z 58.000,A 180.000,B 0.000,C 180.000} C_DIS
LIN {X 73.120,Y 83.586,Z 58.000,A 180.000,B 0.000,C 180.000} C_DIS
LIN {X 72.992,Y 83.489,Z 58.000,A 180.000,B 0.000,C 180.000} C_DIS
LIN {X 72.762,Y 83.310,Z 58.000,A 180.000,B 0.000,C 180.000} C_DIS
LIN {X 72.584,Y 83.158,Z 58.000,A 180.000,B 0.000,C 180.000} C_DIS
LIN {X 72.405,Y 83.000,Z 58.000,A 180.000,B 0.000,C 180.000} C_DIS
LIN {X 72.353,Y 82.952,Z 58.000,A 180.000,B 0.000,C 180.000} C_DIS
LIN {X 72.048,Y 82.647,Z 58.000,A 180.000,B 0.000,C 180.000} C_DIS
LIN {X 72.000,Y 82.595,Z 58.000,A 180.000,B 0.000,C 180.000} C_DIS
LIN {X 71.842,Y 82.416,Z 58.000,A 180.000,B 0.000,C 180.000} C_DIS
LIN {X 71.690,Y 82.238,Z 58.000,A 180.000,B 0.000,C 180.000} C_DIS
LIN {X 71.511,Y 82.008,Z 58.000,A 180.000,B 0.000,C 180.000} C_DIS
LIN {X 71.414,Y 81.880,Z 58.000,A 180.000,B 0.000,C 180.000} C_DIS
LIN {X 71.171,Y 81.522,Z 58.000,A 180.000,B 0.000,C 180.000} C_DIS
LIN {X 71.154,Y 81.493,Z 58.000,A 180.000,B 0.000,C 180.000} C_DIS
LIN {X 70.960,Y 81.165,Z 58.000,A 180.000,B 0.000,C 180.000} C_DIS
LIN {X 70.864,Y 80.986,Z 58.000,A 180.000,B 0.000,C 180.000} C_DIS
LIN {X 70.773,Y 80.807,Z 58.000,A 180.000,B 0.000,C 180.000} C_DIS
LIN {X 70.687,Y 80.628,Z 58.000,A 180.000,B 0.000,C 180.000} C_DIS
LIN {X 70.532,Y 80.271,Z 58.000,A 180.000,B 0.000,C 180.000} C_DIS
LIN {X 70.467,Y 80.092,Z 58.000,A 180.000,B 0.000,C 180.000} C_DIS
LIN {X 70.403,Y 79.913,Z 58.000,A 180.000,B 0.000,C 180.000} C_DIS
LIN {X 70.344,Y 79.735,Z 58.000,A 180.000,B 0.000,C 180.000} C_DIS
LIN {X 70.240,Y 79.377,Z 58.000,A 180.000,B 0.000,C 180.000} C_DIS
LIN {X 70.200,Y 79.198,Z 58.000,A 180.000,B 0.000,C 180.000} C_DIS
LIN {X 70.160,Y 79.020,Z 58.000,A 180.000,B 0.000,C 180.000} C_DIS
LIN {X 70.124,Y 78.841,Z 58.000,A 180.000,B 0.000,C 180.000} C_DIS
LIN {X 70.067,Y 78.483,Z 58.000,A 180.000,B 0.000,C 180.000} C_DIS
LIN {X 70.048,Y 78.304,Z 58.000,A 180.000,B 0.000,C 180.000} C_DIS
LIN {X 70.031,Y 78.126,Z 58.000,A 180.000,B 0.000,C 180.000} C_DIS
LIN {X 70.015,Y 77.947,Z 58.000,A 180.000,B 0.000,C 180.000} C_DIS
LIN {X 70.004,Y 77.589,Z 58.000,A 180.000,B 0.000,C 180.000} C_DIS
LIN {X 70.004,Y 77.411,Z 58.000,A 180.000,B 0.000,C 180.000} C_DIS
LIN {X 70.015,Y 77.053,Z 58.000,A 180.000,B 0.000,C 180.000} C_DIS
LIN {X 70.031,Y 76.874,Z 58.000,A 180.000,B 0.000,C 180.000} C_DIS
LIN {X 70.048,Y 76.696,Z 58.000,A 180.000,B 0.000,C 180.000} C_DIS
LIN {X 70.067,Y 76.517,Z 58.000,A 180.000,B 0.000,C 180.000} C_DIS
LIN {X 70.124,Y 76.159,Z 58.000,A 180.000,B 0.000,C 180.000} C_DIS
LIN {X 70.160,Y 75.980,Z 58.000,A 180.000,B 0.000,C 180.000} C_DIS
LIN {X 70.200,Y 75.802,Z 58.000,A 180.000,B 0.000,C 180.000} C_DIS
LIN {X 70.240,Y 75.623,Z 58.000,A 180.000,B 0.000,C 180.000} C_DIS
LIN {X 70.344,Y 75.265,Z 58.000,A 180.000,B 0.000,C 180.000} C_DIS
LIN {X 70.403,Y 75.087,Z 58.000,A 180.000,B 0.000,C 180.000} C_DIS
LIN {X 70.467,Y 74.908,Z 58.000,A 180.000,B 0.000,C 180.000} C_DIS
LIN {X 70.532,Y 74.729,Z 58.000,A 180.000,B 0.000,C 180.000} C_DIS
LIN {X 70.687,Y 74.372,Z 58.000,A 180.000,B 0.000,C 180.000} C_DIS
LIN {X 70.773,Y 74.193,Z 58.000,A 180.000,B 0.000,C 180.000} C_DIS
LIN {X 70.864,Y 74.014,Z 58.000,A 180.000,B 0.000,C 180.000} C_DIS
LIN {X 70.960,Y 73.835,Z 58.000,A 180.000,B 0.000,C 180.000} C_DIS
LIN {X 71.154,Y 73.507,Z 58.000,A 180.000,B 0.000,C 180.000} C_DIS
LIN {X 71.171,Y 73.478,Z 58.000,A 180.000,B 0.000,C 180.000} C_DIS
LIN {X 71.414,Y 73.120,Z 58.000,A 180.000,B 0.000,C 180.000} C_DIS
LIN {X 71.511,Y 72.992,Z 58.000,A 180.000,B 0.000,C 180.000} C_DIS
LIN {X 71.690,Y 72.762,Z 58.000,A 180.000,B 0.000,C 180.000} C_DIS
LIN {X 71.842,Y 72.584,Z 58.000,A 180.000,B 0.000,C 180.000} C_DIS
LIN {X 72.000,Y 72.405,Z 58.000,A 180.000,B 0.000,C 180.000} C_DIS
LIN {X 72.048,Y 72.353,Z 58.000,A 180.000,B 0.000,C 180.000} C_DIS
LIN {X 72.353,Y 72.048,Z 58.000,A 180.000,B 0.000,C 180.000} C_DIS
LIN {X 72.405,Y 72.000,Z 58.000,A 180.000,B 0.000,C 180.000} C_DIS
LIN {X 72.584,Y 71.842,Z 58.000,A 180.000,B 0.000,C 180.000} C_DIS
LIN {X 72.762,Y 71.690,Z 58.000,A 180.000,B 0.000,C 180.000} C_DIS
LIN {X 72.992,Y 71.511,Z 58.000,A 180.000,B 0.000,C 180.000} C_DIS
LIN {X 73.120,Y 71.414,Z 58.000,A 180.000,B 0.000,C 180.000} C_DIS
LIN {X 73.478,Y 71.171,Z 58.000,A 180.000,B 0.000,C 180.000} C_DIS
LIN {X 73.507,Y 71.154,Z 58.000,A 180.000,B 0.000,C 180.000} C_DIS
LIN {X 73.835,Y 70.960,Z 58.000,A 180.000,B 0.000,C 180.000} C_DIS
LIN {X 74.014,Y 70.864,Z 58.000,A 180.000,B 0.000,C 180.000} C_DIS
LIN {X 74.193,Y 70.773,Z 58.000,A 180.000,B 0.000,C 180.000} C_DIS
LIN {X 74.372,Y 70.687,Z 58.000,A 180.000,B 0.000,C 180.000} C_DIS
LIN {X 74.729,Y 70.532,Z 58.000,A 180.000,B 0.000,C 180.000} C_DIS
LIN {X 74.908,Y 70.467,Z 58.000,A 180.000,B 0.000,C 180.000} C_DIS
LIN {X 75.087,Y 70.403,Z 58.000,A 180.000,B 0.000,C 180.000} C_DIS
LIN {X 75.265,Y 70.344,Z 58.000,A 180.000,B 0.000,C 180.000} C_DIS
LIN {X 75.623,Y 70.240,Z 58.000,A 180.000,B 0.000,C 180.000} C_DIS
LIN {X 75.802,Y 70.200,Z 58.000,A 180.000,B 0.000,C 180.000} C_DIS
LIN {X 75.980,Y 70.160,Z 58.000,A 180.000,B 0.000,C 180.000} C_DIS
LIN {X 76.159,Y 70.124,Z 58.000,A 180.000,B 0.000,C 180.000} C_DIS
LIN {X 76.517,Y 70.067,Z 58.000,A 180.000,B 0.000,C 180.000} C_DIS
LIN {X 76.696,Y 70.048,Z 58.000,A 180.000,B 0.000,C 180.000} C_DIS
LIN {X 76.874,Y 70.031,Z 58.000,A 180.000,B 0.000,C 180.000} C_DIS
LIN {X 77.053,Y 70.015,Z 58.000,A 180.000,B 0.000,C 180.000} C_DIS
LIN {X 77.411,Y 70.004,Z 58.000,A 180.000,B 0.000,C 180.000} C_DIS
LIN {X 77.589,Y 70.004,Z 58.000,A 180.000,B 0.000,C 180.000} C_DIS
LIN {X 77.947,Y 70.015,Z 58.000,A 180.000,B 0.000,C 180.000} C_DIS
LIN {X 78.126,Y 70.031,Z 58.000,A 180.000,B 0.000,C 180.000} C_DIS
LIN {X 78.304,Y 70.048,Z 58.000,A 180.000,B 0.000,C 180.000} C_DIS
LIN {X 78.483,Y 70.067,Z 58.000,A 180.000,B 0.000,C 180.000} C_DIS
LIN {X 78.841,Y 70.124,Z 58.000,A 180.000,B 0.000,C 180.000} C_DIS
LIN {X 79.020,Y 70.160,Z 58.000,A 180.000,B 0.000,C 180.000} C_DIS
LIN {X 79.198,Y 70.200,Z 58.000,A 180.000,B 0.000,C 180.000} C_DIS
LIN {X 79.377,Y 70.240,Z 58.000,A 180.000,B 0.000,C 180.000} C_DIS
LIN {X 79.735,Y 70.344,Z 58.000,A 180.000,B 0.000,C 180.000} C_DIS
LIN {X 79.913,Y 70.403,Z 58.000,A 180.000,B 0.000,C 180.000} C_DIS
LIN {X 80.092,Y 70.467,Z 58.000,A 180.000,B 0.000,C 180.000} C_DIS
LIN {X 80.271,Y 70.532,Z 58.000,A 180.000,B 0.000,C 180.000} C_DIS
LIN {X 80.628,Y 70.687,Z 58.000,A 180.000,B 0.000,C 180.000} C_DIS
LIN {X 80.807,Y 70.773,Z 58.000,A 180.000,B 0.000,C 180.000} C_DIS
LIN {X 80.986,Y 70.864,Z 58.000,A 180.000,B 0.000,C 180.000} C_DIS
LIN {X 81.165,Y 70.960,Z 58.000,A 180.000,B 0.000,C 180.000} C_DIS
LIN {X 81.493,Y 71.154,Z 58.000,A 180.000,B 0.000,C 180.000} C_DIS
LIN {X 81.522,Y 71.171,Z 58.000,A 180.000,B 0.000,C 180.000} C_DIS
LIN {X 81.880,Y 71.414,Z 58.000,A 180.000,B 0.000,C 180.000} C_DIS
LIN {X 82.008,Y 71.511,Z 58.000,A 180.000,B 0.000,C 180.000} C_DIS
LIN {X 82.238,Y 71.690,Z 58.000,A 180.000,B 0.000,C 180.000} C_DIS
LIN {X 82.416,Y 71.842,Z 58.000,A 180.000,B 0.000,C 180.000} C_DIS
LIN {X 82.595,Y 72.000,Z 58.000,A 180.000,B 0.000,C 180.000} C_DIS
LIN {X 82.647,Y 72.048,Z 58.000,A 180.000,B 0.000,C 180.000} C_DIS
LIN {X 82.952,Y 72.353,Z 58.000,A 180.000,B 0.000,C 180.000} C_DIS
LIN {X 83.000,Y 72.405,Z 58.000,A 180.000,B 0.000,C 180.000} C_DIS
LIN {X 83.158,Y 72.584,Z 58.000,A 180.000,B 0.000,C 180.000} C_DIS
LIN {X 83.310,Y 72.762,Z 58.000,A 180.000,B 0.000,C 180.000} C_DIS
LIN {X 83.489,Y 72.992,Z 58.000,A 180.000,B 0.000,C 180.000} C_DIS
LIN {X 83.586,Y 73.120,Z 58.000,A 180.000,B 0.000,C 180.000} C_DIS
LIN {X 83.829,Y 73.478,Z 58.000,A 180.000,B 0.000,C 180.000} C_DIS
LIN {X 83.846,Y 73.507,Z 58.000,A 180.000,B 0.000,C 180.000} C_DIS
LIN {X 84.040,Y 73.835,Z 58.000,A 180.000,B 0.000,C 180.000} C_DIS
LIN {X 84.136,Y 74.014,Z 58.000,A 180.000,B 0.000,C 180.000} C_DIS
LIN {X 84.227,Y 74.193,Z 58.000,A 180.000,B 0.000,C 180.000} C_DIS
LIN {X 84.313,Y 74.372,Z 58.000,A 180.000,B 0.000,C 180.000} C_DIS
LIN {X 84.468,Y 74.729,Z 58.000,A 180.000,B 0.000,C 180.000} C_DIS
LIN {X 84.533,Y 74.908,Z 58.000,A 180.000,B 0.000,C 180.000} C_DIS
LIN {X 84.597,Y 75.087,Z 58.000,A 180.000,B 0.000,C 180.000} C_DIS
LIN {X 84.656,Y 75.265,Z 58.000,A 180.000,B 0.000,C 180.000} C_DIS
LIN {X 84.760,Y 75.623,Z 58.000,A 180.000,B 0.000,C 180.000} C_DIS
LIN {X 84.800,Y 75.802,Z 58.000,A 180.000,B 0.000,C 180.000} C_DIS
LIN {X 84.840,Y 75.980,Z 58.000,A 180.000,B 0.000,C 180.000} C_DIS
LIN {X 84.876,Y 76.159,Z 58.000,A 180.000,B 0.000,C 180.000} C_DIS
LIN {X 84.933,Y 76.517,Z 58.000,A 180.000,B 0.000,C 180.000} C_DIS
LIN {X 84.952,Y 76.696,Z 58.000,A 180.000,B 0.000,C 180.000} C_DIS
LIN {X 84.969,Y 76.874,Z 58.000,A 180.000,B 0.000,C 180.000} C_DIS
LIN {X 84.985,Y 77.053,Z 58.000,A 180.000,B 0.000,C 180.000} C_DIS
LIN {X 84.996,Y 77.411,Z 58.000,A 180.000,B 0.000,C 180.000} C_DIS
LIN {X 84.996,Y 77.589,Z 58.000,A 180.000,B 0.000,C 180.000} C_DIS
LIN {X 84.985,Y 77.947,Z 58.000,A 180.000,B 0.000,C 180.000} C_DIS
LIN {X 84.969,Y 78.126,Z 58.000,A 180.000,B 0.000,C 180.000} C_DIS
LIN {X 84.952,Y 78.304,Z 58.000,A 180.000,B 0.000,C 180.000} C_DIS
LIN {X 84.933,Y 78.483,Z 58.000,A 180.000,B 0.000,C 180.000} C_DIS
LIN {X 84.876,Y 78.841,Z 58.000,A 180.000,B 0.000,C 180.000} C_DIS
LIN {X 84.840,Y 79.020,Z 58.000,A 180.000,B 0.000,C 180.000} C_DIS
LIN {X 84.800,Y 79.198,Z 58.000,A 180.000,B 0.000,C 180.000} C_DIS
LIN {X 84.760,Y 79.377,Z 58.000,A 180.000,B 0.000,C 180.000} C_DIS
LIN {X 84.656,Y 79.735,Z 58.000,A 180.000,B 0.000,C 180.000} C_DIS
LIN {X 84.597,Y 79.913,Z 58.000,A 180.000,B 0.000,C 180.000} C_DIS
LIN {X 84.533,Y 80.092,Z 58.000,A 180.000,B 0.000,C 180.000} C_DIS
LIN {X 84.468,Y 80.271,Z 58.000,A 180.000,B 0.000,C 180.000} C_DIS
LIN {X 84.313,Y 80.628,Z 58.000,A 180.000,B 0.000,C 180.000} C_DIS
LIN {X 84.227,Y 80.807,Z 58.000,A 180.000,B 0.000,C 180.000} C_DIS
LIN {X 84.136,Y 80.986,Z 58.000,A 180.000,B 0.000,C 180.000} C_DIS
LIN {X 84.040,Y 81.165,Z 58.000,A 180.000,B 0.000,C 180.000} C_DIS
LIN {X 83.846,Y 81.493,Z 58.000,A 180.000,B 0.000,C 180.000} C_DIS
LIN {X 83.829,Y 81.522,Z 58.000,A 180.000,B 0.000,C 180.000} C_DIS
LIN {X 83.586,Y 81.880,Z 58.000,A 180.000,B 0.000,C 180.000} C_DIS
LIN {X 83.489,Y 82.008,Z 58.000,A 180.000,B 0.000,C 180.000} C_DIS
LIN {X 83.310,Y 82.238,Z 58.000,A 180.000,B 0.000,C 180.000} C_DIS
LIN {X 83.158,Y 82.416,Z 58.000,A 180.000,B 0.000,C 180.000} C_DIS
LIN {X 83.000,Y 82.595,Z 58.000,A 180.000,B 0.000,C 180.000} C_DIS
LIN {X 82.952,Y 82.647,Z 58.000,A 180.000,B 0.000,C 180.000} C_DIS
LIN {X 82.647,Y 82.952,Z 58.000,A 180.000,B 0.000,C 180.000} C_DIS
LIN {X 82.595,Y 83.000,Z 58.000,A 180.000,B 0.000,C 180.000} C_DIS
LIN {X 82.526,Y 83.061,Z 58.000,A 180.000,B 0.000,C 180.000} C_DIS
; Link Move Starts
LIN {X 82.289,Y 83.270,Z 58.000,A 180.000,B 0.000,C 180.000} C_DIS
LIN {X 82.041,Y 83.463,Z 57.999,A 180.000,B 0.000,C 180.000} C_DIS
LIN {X 81.786,Y 83.649,Z 57.998,A 180.000,B 0.000,C 180.000} C_DIS
LIN {X 81.526,Y 83.826,Z 57.996,A 180.000,B 0.000,C 180.000} C_DIS
LIN {X 81.255,Y 83.987,Z 57.994,A 180.000,B 0.000,C 180.000} C_DIS
LIN {X 80.979,Y 84.139,Z 57.991,A 180.000,B 0.000,C 180.000} C_DIS
LIN {X 80.699,Y 84.282,Z 57.988,A 180.000,B 0.000,C 180.000} C_DIS
LIN {X 80.410,Y 84.408,Z 57.985,A 180.000,B 0.000,C 180.000} C_DIS
LIN {X 80.117,Y 84.524,Z 57.981,A 180.000,B 0.000,C 180.000} C_DIS
LIN {X 79.821,Y 84.631,Z 57.977,A 180.000,B 0.000,C 180.000} C_DIS
LIN {X 79.518,Y 84.719,Z 57.972,A 180.000,B 0.000,C 180.000} C_DIS
LIN {X 79.367,Y 84.763,Z 57.969,A 180.000,B 0.000,C 180.000} C_DIS
LIN {X 79.213,Y 84.797,Z 57.967,A 180.000,B 0.000,C 180.000} C_DIS
LIN {X 79.060,Y 84.831,Z 57.964,A 180.000,B 0.000,C 180.000} C_DIS
LIN {X 78.906,Y 84.866,Z 57.961,A 180.000,B 0.000,C 180.000} C_DIS
LIN {X 78.750,Y 84.890,Z 57.959,A 180.000,B 0.000,C 180.000} C_DIS
LIN {X 78.595,Y 84.915,Z 57.956,A 180.000,B 0.000,C 180.000} C_DIS
LIN {X 78.439,Y 84.940,Z 57.952,A 180.000,B 0.000,C 180.000} C_DIS
LIN {X 78.282,Y 84.955,Z 57.949,A 180.000,B 0.000,C 180.000} C_DIS
LIN {X 78.125,Y 84.969,Z 57.946,A 180.000,B 0.000,C 180.000} C_DIS
LIN {X 77.969,Y 84.984,Z 57.943,A 180.000,B 0.000,C 180.000} C_DIS
LIN {X 77.811,Y 84.989,Z 57.939,A 180.000,B 0.000,C 180.000} C_DIS
LIN {X 77.654,Y 84.994,Z 57.936,A 180.000,B 0.000,C 180.000} C_DIS
LIN {X 77.496,Y 84.999,Z 57.932,A 180.000,B 0.000,C 180.000} C_DIS
LIN {X 77.339,Y 84.994,Z 57.928,A 180.000,B 0.000,C 180.000} C_DIS
LIN {X 77.181,Y 84.989,Z 57.925,A 180.000,B 0.000,C 180.000} C_DIS
LIN {X 77.024,Y 84.983,Z 57.921,A 180.000,B 0.000,C 180.000} C_DIS
LIN {X 76.867,Y 84.969,Z 57.917,A 180.000,B 0.000,C 180.000} C_DIS
LIN {X 76.710,Y 84.954,Z 57.913,A 180.000,B 0.000,C 180.000} C_DIS
LIN {X 76.554,Y 84.939,Z 57.909,A 180.000,B 0.000,C 180.000} C_DIS
LIN {X 76.398,Y 84.914,Z 57.905,A 180.000,B 0.000,C 180.000} C_DIS
LIN {X 76.242,Y 84.889,Z 57.900,A 180.000,B 0.000,C 180.000} C_DIS
LIN {X 76.087,Y 84.864,Z 57.896,A 180.000,B 0.000,C 180.000} C_DIS
LIN {X 75.933,Y 84.830,Z 57.892,A 180.000,B 0.000,C 180.000} C_DIS
LIN {X 75.779,Y 84.795,Z 57.887,A 180.000,B 0.000,C 180.000} C_DIS
LIN {X 75.626,Y 84.760,Z 57.883,A 180.000,B 0.000,C 180.000} C_DIS
LIN {X 75.475,Y 84.717,Z 57.878,A 180.000,B 0.000,C 180.000} C_DIS
LIN {X 75.323,Y 84.673,Z 57.873,A 180.000,B 0.000,C 180.000} C_DIS
LIN {X 75.172,Y 84.628,Z 57.869,A 180.000,B 0.000,C 180.000} C_DIS
LIN {X 75.024,Y 84.575,Z 57.864,A 180.000,B 0.000,C 180.000} C_DIS
LIN {X 74.876,Y 84.521,Z 57.859,A 180.000,B 0.000,C 180.000} C_DIS
LIN {X 74.728,Y 84.467,Z 57.854,A 180.000,B 0.000,C 180.000} C_DIS
LIN {X 74.656,Y 84.436,Z 57.851,A 180.000,B 0.000,C 180.000} C_DIS
LIN {X 74.583,Y 84.405,Z 57.849,A 180.000,B 0.000,C 180.000} C_DIS
LIN {X 74.511,Y 84.373,Z 57.846,A 180.000,B 0.000,C 180.000} C_DIS
LIN {X 74.439,Y 84.342,Z 57.844,A 180.000,B 0.000,C 180.000} C_DIS
LIN {X 74.367,Y 84.311,Z 57.841,A 180.000,B 0.000,C 180.000} C_DIS
LIN {X 74.295,Y 84.279,Z 57.839,A 180.000,B 0.000,C 180.000} C_DIS
LIN {X 74.224,Y 84.243,Z 57.836,A 180.000,B 0.000,C 180.000} C_DIS
LIN {X 74.084,Y 84.171,Z 57.831,A 180.000,B 0.000,C 180.000} C_DIS
LIN {X 73.944,Y 84.100,Z 57.825,A 180.000,B 0.000,C 180.000} C_DIS
LIN {X 73.874,Y 84.063,Z 57.823,A 180.000,B 0.000,C 180.000} C_DIS
LIN {X 73.738,Y 83.983,Z 57.817,A 180.000,B 0.000,C 180.000} C_DIS
LIN {X 73.603,Y 83.903,Z 57.812,A 180.000,B 0.000,C 180.000} C_DIS
LIN {X 73.535,Y 83.863,Z 57.809,A 180.000,B 0.000,C 180.000} C_DIS
LIN {X 73.468,Y 83.822,Z 57.806,A 180.000,B 0.000,C 180.000} C_DIS
LIN {X 73.338,Y 83.733,Z 57.801,A 180.000,B 0.000,C 180.000} C_DIS
LIN {X 73.142,Y 83.601,Z 57.793,A 180.000,B 0.000,C 180.000} C_DIS
LIN {X 73.078,Y 83.555,Z 57.790,A 180.000,B 0.000,C 180.000} C_DIS
LIN {X 72.891,Y 83.410,Z 57.782,A 180.000,B 0.000,C 180.000} C_DIS
LIN {X 72.767,Y 83.314,Z 57.776,A 180.000,B 0.000,C 180.000} C_DIS
LIN {X 72.705,Y 83.265,Z 57.774,A 180.000,B 0.000,C 180.000} C_DIS
LIN {X 72.587,Y 83.161,Z 57.768,A 180.000,B 0.000,C 180.000} C_DIS
LIN {X 72.410,Y 83.004,Z 57.760,A 180.000,B 0.000,C 180.000} C_DIS
LIN {X 72.352,Y 82.951,Z 57.757,A 180.000,B 0.000,C 180.000} C_DIS
LIN {X 72.185,Y 82.784,Z 57.749,A 180.000,B 0.000,C 180.000} C_DIS
LIN {X 72.073,Y 82.673,Z 57.743,A 180.000,B 0.000,C 180.000} C_DIS
LIN {X 72.018,Y 82.616,Z 57.741,A 180.000,B 0.000,C 180.000} C_DIS
LIN {X 71.914,Y 82.498,Z 57.735,A 180.000,B 0.000,C 180.000} C_DIS
LIN {X 71.758,Y 82.321,Z 57.727,A 180.000,B 0.000,C 180.000} C_DIS
LIN {X 71.707,Y 82.261,Z 57.724,A 180.000,B 0.000,C 180.000} C_DIS
LIN {X 71.466,Y 81.949,Z 57.710,A 180.000,B 0.000,C 180.000} C_DIS
LIN {X 71.419,Y 81.886,Z 57.708,A 180.000,B 0.000,C 180.000} C_DIS
LIN {X 71.330,Y 81.756,Z 57.702,A 180.000,B 0.000,C 180.000} C_DIS
LIN {X 71.198,Y 81.561,Z 57.694,A 180.000,B 0.000,C 180.000} C_DIS
LIN {X 71.155,Y 81.495,Z 57.691,A 180.000,B 0.000,C 180.000} C_DIS
LIN {X 70.954,Y 81.156,Z 57.677,A 180.000,B 0.000,C 180.000} C_DIS
LIN {X 70.916,Y 81.087,Z 57.675,A 180.000,B 0.000,C 180.000} C_DIS
LIN {X 70.844,Y 80.947,Z 57.669,A 180.000,B 0.000,C 180.000} C_DIS
LIN {X 70.737,Y 80.736,Z 57.661,A 180.000,B 0.000,C 180.000} C_DIS
LIN {X 70.703,Y 80.665,Z 57.658,A 180.000,B 0.000,C 180.000} C_DIS
LIN {X 70.547,Y 80.304,Z 57.644,A 180.000,B 0.000,C 180.000} C_DIS
LIN {X 70.517,Y 80.231,Z 57.642,A 180.000,B 0.000,C 180.000} C_DIS
LIN {X 70.437,Y 80.008,Z 57.633,A 180.000,B 0.000,C 180.000} C_DIS
LIN {X 70.384,Y 79.860,Z 57.628,A 180.000,B 0.000,C 180.000} C_DIS
LIN {X 70.359,Y 79.785,Z 57.625,A 180.000,B 0.000,C 180.000} C_DIS
LIN {X 70.249,Y 79.407,Z 57.611,A 180.000,B 0.000,C 180.000} C_DIS
LIN {X 70.229,Y 79.331,Z 57.609,A 180.000,B 0.000,C 180.000} C_DIS
LIN {X 70.178,Y 79.100,Z 57.600,A 180.000,B 0.000,C 180.000} C_DIS
LIN {X 70.143,Y 78.947,Z 57.595,A 180.000,B 0.000,C 180.000} C_DIS
LIN {X 70.128,Y 78.869,Z 57.592,A 180.000,B 0.000,C 180.000} C_DIS
LIN {X 70.067,Y 78.480,Z 57.578,A 180.000,B 0.000,C 180.000} C_DIS
LIN {X 70.057,Y 78.402,Z 57.576,A 180.000,B 0.000,C 180.000} C_DIS
LIN {X 70.020,Y 78.010,Z 57.562,A 180.000,B 0.000,C 180.000} C_DIS
LIN {X 70.015,Y 77.932,Z 57.559,A 180.000,B 0.000,C 180.000} C_DIS
LIN {X 70.002,Y 77.538,Z 57.545,A 180.000,B 0.000,C 180.000} C_DIS
LIN {X 70.003,Y 77.459,Z 57.543,A 180.000,B 0.000,C 180.000} C_DIS
LIN {X 70.015,Y 77.066,Z 57.529,A 180.000,B 0.000,C 180.000} C_DIS
LIN {X 70.020,Y 76.987,Z 57.526,A 180.000,B 0.000,C 180.000} C_DIS
LIN {X 70.057,Y 76.595,Z 57.512,A 180.000,B 0.000,C 180.000} C_DIS
LIN {X 70.067,Y 76.517,Z 57.510,A 180.000,B 0.000,C 180.000} C_DIS
LIN {X 70.129,Y 76.128,Z 57.496,A 180.000,B 0.000,C 180.000} C_DIS
LIN {X 70.144,Y 76.051,Z 57.493,A 180.000,B 0.000,C 180.000} C_DIS
LIN {X 70.230,Y 75.667,Z 57.479,A 180.000,B 0.000,C 180.000} C_DIS
LIN {X 70.250,Y 75.590,Z 57.477,A 180.000,B 0.000,C 180.000} C_DIS
LIN {X 70.360,Y 75.212,Z 57.463,A 180.000,B 0.000,C 180.000} C_DIS
LIN {X 70.384,Y 75.138,Z 57.460,A 180.000,B 0.000,C 180.000} C_DIS
LIN {X 70.518,Y 74.767,Z 57.446,A 180.000,B 0.000,C 180.000} C_DIS
LIN {X 70.547,Y 74.694,Z 57.444,A 180.000,B 0.000,C 180.000} C_DIS
LIN {X 70.704,Y 74.333,Z 57.430,A 180.000,B 0.000,C 180.000} C_DIS
LIN {X 70.738,Y 74.262,Z 57.427,A 180.000,B 0.000,C 180.000} C_DIS
LIN {X 70.917,Y 73.911,Z 57.413,A 180.000,B 0.000,C 180.000} C_DIS
LIN {X 70.955,Y 73.842,Z 57.411,A 180.000,B 0.000,C 180.000} C_DIS
LIN {X 71.076,Y 73.639,Z 57.402,A 180.000,B 0.000,C 180.000} C_DIS
LIN {X 71.156,Y 73.503,Z 57.397,A 180.000,B 0.000,C 180.000} C_DIS
LIN {X 71.199,Y 73.437,Z 57.394,A 180.000,B 0.000,C 180.000} C_DIS
LIN {X 71.420,Y 73.112,Z 57.380,A 180.000,B 0.000,C 180.000} C_DIS
LIN {X 71.467,Y 73.049,Z 57.378,A 180.000,B 0.000,C 180.000} C_DIS
LIN {X 71.612,Y 72.862,Z 57.369,A 180.000,B 0.000,C 180.000} C_DIS
LIN {X 71.709,Y 72.737,Z 57.364,A 180.000,B 0.000,C 180.000} C_DIS
LIN {X 71.760,Y 72.677,Z 57.361,A 180.000,B 0.000,C 180.000} C_DIS
LIN {X 72.020,Y 72.382,Z 57.347,A 180.000,B 0.000,C 180.000} C_DIS
LIN {X 72.075,Y 72.326,Z 57.345,A 180.000,B 0.000,C 180.000} C_DIS
LIN {X 72.242,Y 72.159,Z 57.336,A 180.000,B 0.000,C 180.000} C_DIS
LIN {X 72.353,Y 72.047,Z 57.331,A 180.000,B 0.000,C 180.000} C_DIS
LIN {X 72.412,Y 71.994,Z 57.328,A 180.000,B 0.000,C 180.000} C_DIS
LIN {X 72.707,Y 71.734,Z 57.314,A 180.000,B 0.000,C 180.000} C_DIS
LIN {X 72.768,Y 71.685,Z 57.312,A 180.000,B 0.000,C 180.000} C_DIS
LIN {X 72.893,Y 71.588,Z 57.306,A 180.000,B 0.000,C 180.000} C_DIS
LIN {X 73.080,Y 71.443,Z 57.298,A 180.000,B 0.000,C 180.000} C_DIS
LIN {X 73.144,Y 71.398,Z 57.295,A 180.000,B 0.000,C 180.000} C_DIS
LIN {X 73.470,Y 71.177,Z 57.281,A 180.000,B 0.000,C 180.000} C_DIS
LIN {X 73.537,Y 71.136,Z 57.279,A 180.000,B 0.000,C 180.000} C_DIS
LIN {X 73.673,Y 71.056,Z 57.273,A 180.000,B 0.000,C 180.000} C_DIS
LIN {X 73.876,Y 70.936,Z 57.265,A 180.000,B 0.000,C 180.000} C_DIS
LIN {X 73.946,Y 70.899,Z 57.262,A 180.000,B 0.000,C 180.000} C_DIS
LIN {X 74.156,Y 70.792,Z 57.254,A 180.000,B 0.000,C 180.000} C_DIS
LIN {X 74.297,Y 70.720,Z 57.248,A 180.000,B 0.000,C 180.000} C_DIS
LIN {X 74.369,Y 70.688,Z 57.246,A 180.000,B 0.000,C 180.000} C_DIS
LIN {X 74.513,Y 70.626,Z 57.240,A 180.000,B 0.000,C 180.000} C_DIS
LIN {X 74.730,Y 70.532,Z 57.232,A 180.000,B 0.000,C 180.000} C_DIS
LIN {X 74.804,Y 70.505,Z 57.229,A 180.000,B 0.000,C 180.000} C_DIS
LIN {X 75.026,Y 70.425,Z 57.221,A 180.000,B 0.000,C 180.000} C_DIS
LIN {X 75.174,Y 70.371,Z 57.215,A 180.000,B 0.000,C 180.000} C_DIS
LIN {X 75.250,Y 70.349,Z 57.213,A 180.000,B 0.000,C 180.000} C_DIS
LIN {X 75.401,Y 70.305,Z 57.207,A 180.000,B 0.000,C 180.000} C_DIS
LIN {X 75.628,Y 70.239,Z 57.199,A 180.000,B 0.000,C 180.000} C_DIS
LIN {X 75.705,Y 70.221,Z 57.196,A 180.000,B 0.000,C 180.000} C_DIS
LIN {X 75.859,Y 70.187,Z 57.191,A 180.000,B 0.000,C 180.000} C_DIS
LIN {X 76.012,Y 70.153,Z 57.185,A 180.000,B 0.000,C 180.000} C_DIS
LIN {X 76.089,Y 70.135,Z 57.182,A 180.000,B 0.000,C 180.000} C_DIS
LIN {X 76.167,Y 70.123,Z 57.180,A 180.000,B 0.000,C 180.000} C_DIS
LIN {X 76.322,Y 70.098,Z 57.174,A 180.000,B 0.000,C 180.000} C_DIS
LIN {X 76.478,Y 70.073,Z 57.169,A 180.000,B 0.000,C 180.000} C_DIS
LIN {X 76.556,Y 70.061,Z 57.166,A 180.000,B 0.000,C 180.000} C_DIS
LIN {X 76.634,Y 70.053,Z 57.164,A 180.000,B 0.000,C 180.000} C_DIS
LIN {X 76.713,Y 70.046,Z 57.161,A 180.000,B 0.000,C 180.000} C_DIS
LIN {X 76.791,Y 70.039,Z 57.159,A 180.000,B 0.000,C 180.000} C_DIS
LIN {X 76.869,Y 70.031,Z 57.156,A 180.000,B 0.000,C 180.000} C_DIS
LIN {X 76.948,Y 70.024,Z 57.154,A 180.000,B 0.000,C 180.000} C_DIS
LIN {X 77.026,Y 70.016,Z 57.151,A 180.000,B 0.000,C 180.000} C_DIS
LIN {X 77.105,Y 70.014,Z 57.149,A 180.000,B 0.000,C 180.000} C_DIS
LIN {X 77.262,Y 70.009,Z 57.144,A 180.000,B 0.000,C 180.000} C_DIS
LIN {X 77.420,Y 70.004,Z 57.139,A 180.000,B 0.000,C 180.000} C_DIS
LIN {X 77.577,Y 70.004,Z 57.134,A 180.000,B 0.000,C 180.000} C_DIS
LIN {X 77.735,Y 70.009,Z 57.129,A 180.000,B 0.000,C 180.000} C_DIS
LIN {X 77.892,Y 70.014,Z 57.124,A 180.000,B 0.000,C 180.000} C_DIS
LIN {X 78.049,Y 70.023,Z 57.120,A 180.000,B 0.000,C 180.000} C_DIS
LIN {X 78.206,Y 70.038,Z 57.115,A 180.000,B 0.000,C 180.000} C_DIS
LIN {X 78.363,Y 70.053,Z 57.111,A 180.000,B 0.000,C 180.000} C_DIS
LIN {X 78.519,Y 70.073,Z 57.106,A 180.000,B 0.000,C 180.000} C_DIS
LIN {X 78.675,Y 70.098,Z 57.102,A 180.000,B 0.000,C 180.000} C_DIS
LIN {X 78.830,Y 70.122,Z 57.097,A 180.000,B 0.000,C 180.000} C_DIS
LIN {X 78.985,Y 70.152,Z 57.093,A 180.000,B 0.000,C 180.000} C_DIS
LIN {X 79.139,Y 70.186,Z 57.089,A 180.000,B 0.000,C 180.000} C_DIS
LIN {X 79.292,Y 70.221,Z 57.085,A 180.000,B 0.000,C 180.000} C_DIS
LIN {X 79.445,Y 70.260,Z 57.081,A 180.000,B 0.000,C 180.000} C_DIS
LIN {X 79.596,Y 70.304,Z 57.077,A 180.000,B 0.000,C 180.000} C_DIS
LIN {X 79.747,Y 70.348,Z 57.073,A 180.000,B 0.000,C 180.000} C_DIS
LIN {X 79.897,Y 70.397,Z 57.070,A 180.000,B 0.000,C 180.000} C_DIS
LIN {X 80.045,Y 70.450,Z 57.066,A 180.000,B 0.000,C 180.000} C_DIS
LIN {X 80.193,Y 70.504,Z 57.062,A 180.000,B 0.000,C 180.000} C_DIS
LIN {X 80.340,Y 70.562,Z 57.059,A 180.000,B 0.000,C 180.000} C_DIS
LIN {X 80.484,Y 70.625,Z 57.056,A 180.000,B 0.000,C 180.000} C_DIS
LIN {X 80.629,Y 70.687,Z 57.052,A 180.000,B 0.000,C 180.000} C_DIS
LIN {X 80.771,Y 70.755,Z 57.049,A 180.000,B 0.000,C 180.000} C_DIS
LIN {X 80.911,Y 70.826,Z 57.046,A 180.000,B 0.000,C 180.000} C_DIS
LIN {X 81.052,Y 70.898,Z 57.043,A 180.000,B 0.000,C 180.000} C_DIS
LIN {X 81.189,Y 70.974,Z 57.040,A 180.000,B 0.000,C 180.000} C_DIS
LIN {X 81.325,Y 71.054,Z 57.037,A 180.000,B 0.000,C 180.000} C_DIS
LIN {X 81.460,Y 71.135,Z 57.034,A 180.000,B 0.000,C 180.000} C_DIS
LIN {X 81.593,Y 71.220,Z 57.032,A 180.000,B 0.000,C 180.000} C_DIS
LIN {X 81.723,Y 71.308,Z 57.029,A 180.000,B 0.000,C 180.000} C_DIS
LIN {X 81.854,Y 71.397,Z 57.027,A 180.000,B 0.000,C 180.000} C_DIS
LIN {X 82.105,Y 71.586,Z 57.022,A 180.000,B 0.000,C 180.000} C_DIS
LIN {X 82.350,Y 71.784,Z 57.018,A 180.000,B 0.000,C 180.000} C_DIS
LIN {X 82.586,Y 71.992,Z 57.014,A 180.000,B 0.000,C 180.000} C_DIS
LIN {X 82.812,Y 72.212,Z 57.011,A 180.000,B 0.000,C 180.000} C_DIS
LIN {X 83.030,Y 72.439,Z 57.008,A 180.000,B 0.000,C 180.000} C_DIS
LIN {X 83.238,Y 72.675,Z 57.005,A 180.000,B 0.000,C 180.000} C_DIS
LIN {X 83.434,Y 72.922,Z 57.003,A 180.000,B 0.000,C 180.000} C_DIS
LIN {X 83.623,Y 73.175,Z 57.002,A 180.000,B 0.000,C 180.000} C_DIS
LIN {X 83.800,Y 73.435,Z 57.001,A 180.000,B 0.000,C 180.000} C_DIS
LIN {X 83.963,Y 73.704,Z 57.000,A 180.000,B 0.000,C 180.000} C_DIS
LIN {X 84.078,Y 73.907,Z 57.000,A 180.000,B 0.000,C 180.000} C_DIS
; Cutting Move Starts
LIN {X 84.136,Y 74.014,Z 57.000,A 180.000,B 0.000,C 180.000} C_DIS
LIN {X 84.227,Y 74.193,Z 57.000,A 180.000,B 0.000,C 180.000} C_DIS
LIN {X 84.313,Y 74.372,Z 57.000,A 180.000,B 0.000,C 180.000} C_DIS
LIN {X 84.468,Y 74.729,Z 57.000,A 180.000,B 0.000,C 180.000} C_DIS
LIN {X 84.533,Y 74.908,Z 57.000,A 180.000,B 0.000,C 180.000} C_DIS
LIN {X 84.597,Y 75.087,Z 57.000,A 180.000,B 0.000,C 180.000} C_DIS
LIN {X 84.656,Y 75.265,Z 57.000,A 180.000,B 0.000,C 180.000} C_DIS
LIN {X 84.760,Y 75.623,Z 57.000,A 180.000,B 0.000,C 180.000} C_DIS
LIN {X 84.800,Y 75.802,Z 57.000,A 180.000,B 0.000,C 180.000} C_DIS
LIN {X 84.840,Y 75.980,Z 57.000,A 180.000,B 0.000,C 180.000} C_DIS
LIN {X 84.876,Y 76.159,Z 57.000,A 180.000,B 0.000,C 180.000} C_DIS
LIN {X 84.933,Y 76.517,Z 57.000,A 180.000,B 0.000,C 180.000} C_DIS
LIN {X 84.952,Y 76.696,Z 57.000,A 180.000,B 0.000,C 180.000} C_DIS
LIN {X 84.969,Y 76.874,Z 57.000,A 180.000,B 0.000,C 180.000} C_DIS
LIN {X 84.985,Y 77.053,Z 57.000,A 180.000,B 0.000,C 180.000} C_DIS
LIN {X 84.996,Y 77.411,Z 57.000,A 180.000,B 0.000,C 180.000} C_DIS
LIN {X 84.996,Y 77.589,Z 57.000,A 180.000,B 0.000,C 180.000} C_DIS
LIN {X 84.985,Y 77.947,Z 57.000,A 180.000,B 0.000,C 180.000} C_DIS
LIN {X 84.969,Y 78.126,Z 57.000,A 180.000,B 0.000,C 180.000} C_DIS
LIN {X 84.952,Y 78.304,Z 57.000,A 180.000,B 0.000,C 180.000} C_DIS
LIN {X 84.933,Y 78.483,Z 57.000,A 180.000,B 0.000,C 180.000} C_DIS
LIN {X 84.876,Y 78.841,Z 57.000,A 180.000,B 0.000,C 180.000} C_DIS
LIN {X 84.840,Y 79.020,Z 57.000,A 180.000,B 0.000,C 180.000} C_DIS
LIN {X 84.800,Y 79.198,Z 57.000,A 180.000,B 0.000,C 180.000} C_DIS
LIN {X 84.760,Y 79.377,Z 57.000,A 180.000,B 0.000,C 180.000} C_DIS
LIN {X 84.656,Y 79.735,Z 57.000,A 180.000,B 0.000,C 180.000} C_DIS
LIN {X 84.597,Y 79.913,Z 57.000,A 180.000,B 0.000,C 180.000} C_DIS
LIN {X 84.533,Y 80.092,Z 57.000,A 180.000,B 0.000,C 180.000} C_DIS
LIN {X 84.468,Y 80.271,Z 57.000,A 180.000,B 0.000,C 180.000} C_DIS
LIN {X 84.313,Y 80.628,Z 57.000,A 180.000,B 0.000,C 180.000} C_DIS
LIN {X 84.227,Y 80.807,Z 57.000,A 180.000,B 0.000,C 180.000} C_DIS
LIN {X 84.136,Y 80.986,Z 57.000,A 180.000,B 0.000,C 180.000} C_DIS
LIN {X 84.040,Y 81.165,Z 57.000,A 180.000,B 0.000,C 180.000} C_DIS
LIN {X 83.846,Y 81.493,Z 57.000,A 180.000,B 0.000,C 180.000} C_DIS
LIN {X 83.829,Y 81.522,Z 57.000,A 180.000,B 0.000,C 180.000} C_DIS
LIN {X 83.586,Y 81.880,Z 57.000,A 180.000,B 0.000,C 180.000} C_DIS
LIN {X 83.489,Y 82.008,Z 57.000,A 180.000,B 0.000,C 180.000} C_DIS
LIN {X 83.310,Y 82.238,Z 57.000,A 180.000,B 0.000,C 180.000} C_DIS
LIN {X 83.158,Y 82.416,Z 57.000,A 180.000,B 0.000,C 180.000} C_DIS
LIN {X 83.000,Y 82.595,Z 57.000,A 180.000,B 0.000,C 180.000} C_DIS
LIN {X 82.952,Y 82.647,Z 57.000,A 180.000,B 0.000,C 180.000} C_DIS
LIN {X 82.647,Y 82.952,Z 57.000,A 180.000,B 0.000,C 180.000} C_DIS
LIN {X 82.595,Y 83.000,Z 57.000,A 180.000,B 0.000,C 180.000} C_DIS
LIN {X 82.416,Y 83.158,Z 57.000,A 180.000,B 0.000,C 180.000} C_DIS
LIN {X 82.238,Y 83.310,Z 57.000,A 180.000,B 0.000,C 180.000} C_DIS
LIN {X 82.008,Y 83.489,Z 57.000,A 180.000,B 0.000,C 180.000} C_DIS
LIN {X 81.880,Y 83.586,Z 57.000,A 180.000,B 0.000,C 180.000} C_DIS
LIN {X 81.522,Y 83.829,Z 57.000,A 180.000,B 0.000,C 180.000} C_DIS
LIN {X 81.493,Y 83.846,Z 57.000,A 180.000,B 0.000,C 180.000} C_DIS
LIN {X 81.165,Y 84.040,Z 57.000,A 180.000,B 0.000,C 180.000} C_DIS
LIN {X 80.986,Y 84.136,Z 57.000,A 180.000,B 0.000,C 180.000} C_DIS
LIN {X 80.807,Y 84.227,Z 57.000,A 180.000,B 0.000,C 180.000} C_DIS
LIN {X 80.628,Y 84.313,Z 57.000,A 180.000,B 0.000,C 180.000} C_DIS
LIN {X 80.271,Y 84.468,Z 57.000,A 180.000,B 0.000,C 180.000} C_DIS
LIN {X 80.092,Y 84.533,Z 57.000,A 180.000,B 0.000,C 180.000} C_DIS
LIN {X 79.913,Y 84.597,Z 57.000,A 180.000,B 0.000,C 180.000} C_DIS
LIN {X 79.735,Y 84.656,Z 57.000,A 180.000,B 0.000,C 180.000} C_DIS
LIN {X 79.377,Y 84.760,Z 57.000,A 180.000,B 0.000,C 180.000} C_DIS
LIN {X 79.198,Y 84.800,Z 57.000,A 180.000,B 0.000,C 180.000} C_DIS
LIN {X 79.020,Y 84.840,Z 57.000,A 180.000,B 0.000,C 180.000} C_DIS
LIN {X 78.841,Y 84.876,Z 57.000,A 180.000,B 0.000,C 180.000} C_DIS
LIN {X 78.483,Y 84.933,Z 57.000,A 180.000,B 0.000,C 180.000} C_DIS
LIN {X 78.304,Y 84.952,Z 57.000,A 180.000,B 0.000,C 180.000} C_DIS
LIN {X 78.126,Y 84.969,Z 57.000,A 180.000,B 0.000,C 180.000} C_DIS
LIN {X 77.947,Y 84.985,Z 57.000,A 180.000,B 0.000,C 180.000} C_DIS
LIN {X 77.589,Y 84.996,Z 57.000,A 180.000,B 0.000,C 180.000} C_DIS
LIN {X 77.411,Y 84.996,Z 57.000,A 180.000,B 0.000,C 180.000} C_DIS
LIN {X 77.053,Y 84.985,Z 57.000,A 180.000,B 0.000,C 180.000} C_DIS
LIN {X 76.874,Y 84.969,Z 57.000,A 180.000,B 0.000,C 180.000} C_DIS
LIN {X 76.696,Y 84.952,Z 57.000,A 180.000,B 0.000,C 180.000} C_DIS
LIN {X 76.517,Y 84.933,Z 57.000,A 180.000,B 0.000,C 180.000} C_DIS
LIN {X 76.159,Y 84.876,Z 57.000,A 180.000,B 0.000,C 180.000} C_DIS
LIN {X 75.980,Y 84.840,Z 57.000,A 180.000,B 0.000,C 180.000} C_DIS
LIN {X 75.802,Y 84.800,Z 57.000,A 180.000,B 0.000,C 180.000} C_DIS
LIN {X 75.623,Y 84.760,Z 57.000,A 180.000,B 0.000,C 180.000} C_DIS
LIN {X 75.265,Y 84.656,Z 57.000,A 180.000,B 0.000,C 180.000} C_DIS
LIN {X 75.087,Y 84.597,Z 57.000,A 180.000,B 0.000,C 180.000} C_DIS
LIN {X 74.908,Y 84.533,Z 57.000,A 180.000,B 0.000,C 180.000} C_DIS
LIN {X 74.729,Y 84.468,Z 57.000,A 180.000,B 0.000,C 180.000} C_DIS
LIN {X 74.372,Y 84.313,Z 57.000,A 180.000,B 0.000,C 180.000} C_DIS
LIN {X 74.193,Y 84.227,Z 57.000,A 180.000,B 0.000,C 180.000} C_DIS
LIN {X 74.014,Y 84.136,Z 57.000,A 180.000,B 0.000,C 180.000} C_DIS
LIN {X 73.835,Y 84.040,Z 57.000,A 180.000,B 0.000,C 180.000} C_DIS
LIN {X 73.507,Y 83.846,Z 57.000,A 180.000,B 0.000,C 180.000} C_DIS
LIN {X 73.478,Y 83.829,Z 57.000,A 180.000,B 0.000,C 180.000} C_DIS
LIN {X 73.120,Y 83.586,Z 57.000,A 180.000,B 0.000,C 180.000} C_DIS
LIN {X 72.992,Y 83.489,Z 57.000,A 180.000,B 0.000,C 180.000} C_DIS
LIN {X 72.762,Y 83.310,Z 57.000,A 180.000,B 0.000,C 180.000} C_DIS
LIN {X 72.584,Y 83.158,Z 57.000,A 180.000,B 0.000,C 180.000} C_DIS
LIN {X 72.405,Y 83.000,Z 57.000,A 180.000,B 0.000,C 180.000} C_DIS
LIN {X 72.353,Y 82.952,Z 57.000,A 180.000,B 0.000,C 180.000} C_DIS
LIN {X 72.048,Y 82.647,Z 57.000,A 180.000,B 0.000,C 180.000} C_DIS
LIN {X 72.000,Y 82.595,Z 57.000,A 180.000,B 0.000,C 180.000} C_DIS
LIN {X 71.842,Y 82.416,Z 57.000,A 180.000,B 0.000,C 180.000} C_DIS
LIN {X 71.690,Y 82.238,Z 57.000,A 180.000,B 0.000,C 180.000} C_DIS
LIN {X 71.511,Y 82.008,Z 57.000,A 180.000,B 0.000,C 180.000} C_DIS
LIN {X 71.414,Y 81.880,Z 57.000,A 180.000,B 0.000,C 180.000} C_DIS
LIN {X 71.171,Y 81.522,Z 57.000,A 180.000,B 0.000,C 180.000} C_DIS
LIN {X 71.154,Y 81.493,Z 57.000,A 180.000,B 0.000,C 180.000} C_DIS
LIN {X 70.960,Y 81.165,Z 57.000,A 180.000,B 0.000,C 180.000} C_DIS
LIN {X 70.864,Y 80.986,Z 57.000,A 180.000,B 0.000,C 180.000} C_DIS
LIN {X 70.773,Y 80.807,Z 57.000,A 180.000,B 0.000,C 180.000} C_DIS
LIN {X 70.687,Y 80.628,Z 57.000,A 180.000,B 0.000,C 180.000} C_DIS
LIN {X 70.532,Y 80.271,Z 57.000,A 180.000,B 0.000,C 180.000} C_DIS
LIN {X 70.467,Y 80.092,Z 57.000,A 180.000,B 0.000,C 180.000} C_DIS
LIN {X 70.403,Y 79.913,Z 57.000,A 180.000,B 0.000,C 180.000} C_DIS
LIN {X 70.344,Y 79.735,Z 57.000,A 180.000,B 0.000,C 180.000} C_DIS
LIN {X 70.240,Y 79.377,Z 57.000,A 180.000,B 0.000,C 180.000} C_DIS
LIN {X 70.200,Y 79.198,Z 57.000,A 180.000,B 0.000,C 180.000} C_DIS
LIN {X 70.160,Y 79.020,Z 57.000,A 180.000,B 0.000,C 180.000} C_DIS
LIN {X 70.124,Y 78.841,Z 57.000,A 180.000,B 0.000,C 180.000} C_DIS
LIN {X 70.067,Y 78.483,Z 57.000,A 180.000,B 0.000,C 180.000} C_DIS
LIN {X 70.048,Y 78.304,Z 57.000,A 180.000,B 0.000,C 180.000} C_DIS
LIN {X 70.031,Y 78.126,Z 57.000,A 180.000,B 0.000,C 180.000} C_DIS
LIN {X 70.015,Y 77.947,Z 57.000,A 180.000,B 0.000,C 180.000} C_DIS
LIN {X 70.004,Y 77.589,Z 57.000,A 180.000,B 0.000,C 180.000} C_DIS
LIN {X 70.004,Y 77.411,Z 57.000,A 180.000,B 0.000,C 180.000} C_DIS
LIN {X 70.015,Y 77.053,Z 57.000,A 180.000,B 0.000,C 180.000} C_DIS
LIN {X 70.031,Y 76.874,Z 57.000,A 180.000,B 0.000,C 180.000} C_DIS
LIN {X 70.048,Y 76.696,Z 57.000,A 180.000,B 0.000,C 180.000} C_DIS
LIN {X 70.067,Y 76.517,Z 57.000,A 180.000,B 0.000,C 180.000} C_DIS
LIN {X 70.124,Y 76.159,Z 57.000,A 180.000,B 0.000,C 180.000} C_DIS
LIN {X 70.160,Y 75.980,Z 57.000,A 180.000,B 0.000,C 180.000} C_DIS
LIN {X 70.200,Y 75.802,Z 57.000,A 180.000,B 0.000,C 180.000} C_DIS
LIN {X 70.240,Y 75.623,Z 57.000,A 180.000,B 0.000,C 180.000} C_DIS
LIN {X 70.344,Y 75.265,Z 57.000,A 180.000,B 0.000,C 180.000} C_DIS
LIN {X 70.403,Y 75.087,Z 57.000,A 180.000,B 0.000,C 180.000} C_DIS
LIN {X 70.467,Y 74.908,Z 57.000,A 180.000,B 0.000,C 180.000} C_DIS
LIN {X 70.532,Y 74.729,Z 57.000,A 180.000,B 0.000,C 180.000} C_DIS
LIN {X 70.687,Y 74.372,Z 57.000,A 180.000,B 0.000,C 180.000} C_DIS
LIN {X 70.773,Y 74.193,Z 57.000,A 180.000,B 0.000,C 180.000} C_DIS
LIN {X 70.864,Y 74.014,Z 57.000,A 180.000,B 0.000,C 180.000} C_DIS
LIN {X 70.960,Y 73.835,Z 57.000,A 180.000,B 0.000,C 180.000} C_DIS
LIN {X 71.154,Y 73.507,Z 57.000,A 180.000,B 0.000,C 180.000} C_DIS
LIN {X 71.171,Y 73.478,Z 57.000,A 180.000,B 0.000,C 180.000} C_DIS
LIN {X 71.414,Y 73.120,Z 57.000,A 180.000,B 0.000,C 180.000} C_DIS
LIN {X 71.511,Y 72.992,Z 57.000,A 180.000,B 0.000,C 180.000} C_DIS
LIN {X 71.690,Y 72.762,Z 57.000,A 180.000,B 0.000,C 180.000} C_DIS
LIN {X 71.842,Y 72.584,Z 57.000,A 180.000,B 0.000,C 180.000} C_DIS
LIN {X 72.000,Y 72.405,Z 57.000,A 180.000,B 0.000,C 180.000} C_DIS
LIN {X 72.048,Y 72.353,Z 57.000,A 180.000,B 0.000,C 180.000} C_DIS
LIN {X 72.353,Y 72.048,Z 57.000,A 180.000,B 0.000,C 180.000} C_DIS
LIN {X 72.405,Y 72.000,Z 57.000,A 180.000,B 0.000,C 180.000} C_DIS
LIN {X 72.584,Y 71.842,Z 57.000,A 180.000,B 0.000,C 180.000} C_DIS
LIN {X 72.762,Y 71.690,Z 57.000,A 180.000,B 0.000,C 180.000} C_DIS
LIN {X 72.992,Y 71.511,Z 57.000,A 180.000,B 0.000,C 180.000} C_DIS
LIN {X 73.120,Y 71.414,Z 57.000,A 180.000,B 0.000,C 180.000} C_DIS
LIN {X 73.478,Y 71.171,Z 57.000,A 180.000,B 0.000,C 180.000} C_DIS
LIN {X 73.507,Y 71.154,Z 57.000,A 180.000,B 0.000,C 180.000} C_DIS
LIN {X 73.835,Y 70.960,Z 57.000,A 180.000,B 0.000,C 180.000} C_DIS
LIN {X 74.014,Y 70.864,Z 57.000,A 180.000,B 0.000,C 180.000} C_DIS
LIN {X 74.193,Y 70.773,Z 57.000,A 180.000,B 0.000,C 180.000} C_DIS
LIN {X 74.372,Y 70.687,Z 57.000,A 180.000,B 0.000,C 180.000} C_DIS
LIN {X 74.729,Y 70.532,Z 57.000,A 180.000,B 0.000,C 180.000} C_DIS
LIN {X 74.908,Y 70.467,Z 57.000,A 180.000,B 0.000,C 180.000} C_DIS
LIN {X 75.087,Y 70.403,Z 57.000,A 180.000,B 0.000,C 180.000} C_DIS
LIN {X 75.265,Y 70.344,Z 57.000,A 180.000,B 0.000,C 180.000} C_DIS
LIN {X 75.623,Y 70.240,Z 57.000,A 180.000,B 0.000,C 180.000} C_DIS
LIN {X 75.802,Y 70.200,Z 57.000,A 180.000,B 0.000,C 180.000} C_DIS
LIN {X 75.980,Y 70.160,Z 57.000,A 180.000,B 0.000,C 180.000} C_DIS
LIN {X 76.159,Y 70.124,Z 57.000,A 180.000,B 0.000,C 180.000} C_DIS
LIN {X 76.517,Y 70.067,Z 57.000,A 180.000,B 0.000,C 180.000} C_DIS
LIN {X 76.696,Y 70.048,Z 57.000,A 180.000,B 0.000,C 180.000} C_DIS
LIN {X 76.874,Y 70.031,Z 57.000,A 180.000,B 0.000,C 180.000} C_DIS
LIN {X 77.053,Y 70.015,Z 57.000,A 180.000,B 0.000,C 180.000} C_DIS
LIN {X 77.411,Y 70.004,Z 57.000,A 180.000,B 0.000,C 180.000} C_DIS
LIN {X 77.589,Y 70.004,Z 57.000,A 180.000,B 0.000,C 180.000} C_DIS
LIN {X 77.947,Y 70.015,Z 57.000,A 180.000,B 0.000,C 180.000} C_DIS
LIN {X 78.126,Y 70.031,Z 57.000,A 180.000,B 0.000,C 180.000} C_DIS
LIN {X 78.304,Y 70.048,Z 57.000,A 180.000,B 0.000,C 180.000} C_DIS
LIN {X 78.483,Y 70.067,Z 57.000,A 180.000,B 0.000,C 180.000} C_DIS
LIN {X 78.841,Y 70.124,Z 57.000,A 180.000,B 0.000,C 180.000} C_DIS
LIN {X 79.020,Y 70.160,Z 57.000,A 180.000,B 0.000,C 180.000} C_DIS
LIN {X 79.198,Y 70.200,Z 57.000,A 180.000,B 0.000,C 180.000} C_DIS
LIN {X 79.377,Y 70.240,Z 57.000,A 180.000,B 0.000,C 180.000} C_DIS
LIN {X 79.735,Y 70.344,Z 57.000,A 180.000,B 0.000,C 180.000} C_DIS
LIN {X 79.913,Y 70.403,Z 57.000,A 180.000,B 0.000,C 180.000} C_DIS
LIN {X 80.092,Y 70.467,Z 57.000,A 180.000,B 0.000,C 180.000} C_DIS
LIN {X 80.271,Y 70.532,Z 57.000,A 180.000,B 0.000,C 180.000} C_DIS
LIN {X 80.628,Y 70.687,Z 57.000,A 180.000,B 0.000,C 180.000} C_DIS
LIN {X 80.807,Y 70.773,Z 57.000,A 180.000,B 0.000,C 180.000} C_DIS
LIN {X 80.986,Y 70.864,Z 57.000,A 180.000,B 0.000,C 180.000} C_DIS
LIN {X 81.165,Y 70.960,Z 57.000,A 180.000,B 0.000,C 180.000} C_DIS
LIN {X 81.493,Y 71.154,Z 57.000,A 180.000,B 0.000,C 180.000} C_DIS
LIN {X 81.522,Y 71.171,Z 57.000,A 180.000,B 0.000,C 180.000} C_DIS
LIN {X 81.880,Y 71.414,Z 57.000,A 180.000,B 0.000,C 180.000} C_DIS
LIN {X 82.008,Y 71.511,Z 57.000,A 180.000,B 0.000,C 180.000} C_DIS
LIN {X 82.238,Y 71.690,Z 57.000,A 180.000,B 0.000,C 180.000} C_DIS
LIN {X 82.416,Y 71.842,Z 57.000,A 180.000,B 0.000,C 180.000} C_DIS
LIN {X 82.595,Y 72.000,Z 57.000,A 180.000,B 0.000,C 180.000} C_DIS
LIN {X 82.647,Y 72.048,Z 57.000,A 180.000,B 0.000,C 180.000} C_DIS
LIN {X 82.952,Y 72.353,Z 57.000,A 180.000,B 0.000,C 180.000} C_DIS
LIN {X 83.000,Y 72.405,Z 57.000,A 180.000,B 0.000,C 180.000} C_DIS
LIN {X 83.158,Y 72.584,Z 57.000,A 180.000,B 0.000,C 180.000} C_DIS
LIN {X 83.310,Y 72.762,Z 57.000,A 180.000,B 0.000,C 180.000} C_DIS
LIN {X 83.489,Y 72.992,Z 57.000,A 180.000,B 0.000,C 180.000} C_DIS
LIN {X 83.586,Y 73.120,Z 57.000,A 180.000,B 0.000,C 180.000} C_DIS
LIN {X 83.829,Y 73.478,Z 57.000,A 180.000,B 0.000,C 180.000} C_DIS
LIN {X 83.846,Y 73.507,Z 57.000,A 180.000,B 0.000,C 180.000} C_DIS
LIN {X 84.040,Y 73.835,Z 57.000,A 180.000,B 0.000,C 180.000} C_DIS
LIN {X 84.078,Y 73.907,Z 57.000,A 180.000,B 0.000,C 180.000} C_DIS
; Lead Out Move Starts
LIN {X 84.084,Y 74.366,Z 57.000,A 180.000,B 0.000,C 180.000} C_DIS
LIN {X 83.712,Y 74.636,Z 57.000,A 180.000,B 0.000,C 180.000} C_DIS
LIN {X 82.807,Y 74.773,Z 57.000,A 180.000,B 0.000,C 180.000} C_DIS
LIN {X 82.458,Y 74.826,Z 57.146,A 180.000,B 0.000,C 180.000} C_DIS
LIN {X 82.313,Y 74.848,Z 57.500,A 180.000,B 0.000,C 180.000} C_DIS
; Rapid Move Starts
LIN {X 82.313,Y 74.848,Z 95.000,A 180.000,B 0.000,C 180.000} C_DIS
LIN {X 114.551,Y 44.141,Z 95.000,A 180.000,B 0.000,C 180.000} C_DIS
LIN {X 114.551,Y 44.141,Z 63.498,A 180.000,B 0.000,C 180.000} C_DIS
; Plunge Move Starts
$VEL.CP=0.01
LIN {X 114.551,Y 44.141,Z 62.625,A 180.000,B 0.000,C 180.000} C_DIS
; Lead In Move Starts
LIN {X 114.551,Y 44.141,Z 61.500,A 180.000,B 0.000,C 180.000} C_DIS
LIN {X 114.447,Y 44.245,Z 61.146,A 180.000,B 0.000,C 180.000} C_DIS
LIN {X 114.197,Y 44.495,Z 61.000,A 180.000,B 0.000,C 180.000} C_DIS
LIN {X 113.967,Y 44.725,Z 61.000,A 180.000,B 0.000,C 180.000} C_DIS
LIN {X 113.614,Y 44.871,Z 61.000,A 180.000,B 0.000,C 180.000} C_DIS
LIN {X 113.260,Y 44.725,Z 61.000,A 180.000,B 0.000,C 180.000} C_DIS
; Cutting Move Starts
$VEL.CP=0.02
LIN {X 79.265,Y 10.729,Z 61.000,A 180.000,B 0.000,C 180.000} C_DIS
LIN {X 79.198,Y 10.665,Z 61.000,A 180.000,B 0.000,C 180.000} C_DIS
LIN {X 79.065,Y 10.551,Z 61.000,A 180.000,B 0.000,C 180.000} C_DIS
LIN {X 79.020,Y 10.515,Z 61.000,A 180.000,B 0.000,C 180.000} C_DIS
LIN {X 78.841,Y 10.390,Z 61.000,A 180.000,B 0.000,C 180.000} C_DIS
LIN {X 78.812,Y 10.372,Z 61.000,A 180.000,B 0.000,C 180.000} C_DIS
LIN {X 78.662,Y 10.286,Z 61.000,A 180.000,B 0.000,C 180.000} C_DIS
LIN {X 78.483,Y 10.201,Z 61.000,A 180.000,B 0.000,C 180.000} C_DIS
LIN {X 78.463,Y 10.193,Z 61.000,A 180.000,B 0.000,C 180.000} C_DIS
LIN {X 78.304,Y 10.133,Z 61.000,A 180.000,B 0.000,C 180.000} C_DIS
LIN {X 78.126,Y 10.080,Z 61.000,A 180.000,B 0.000,C 180.000} C_DIS
LIN {X 77.947,Y 10.040,Z 61.000,A 180.000,B 0.000,C 180.000} C_DIS
LIN {X 77.768,Y 10.014,Z 61.000,A 180.000,B 0.000,C 180.000} C_DIS
LIN {X 77.767,Y 10.014,Z 61.000,A 180.000,B 0.000,C 180.000} C_DIS
LIN {X 77.589,Y 10.002,Z 61.000,A 180.000,B 0.000,C 180.000} C_DIS
LIN {X 77.411,Y 10.002,Z 61.000,A 180.000,B 0.000,C 180.000} C_DIS
LIN {X 77.233,Y 10.014,Z 61.000,A 180.000,B 0.000,C 180.000} C_DIS
LIN {X 77.232,Y 10.014,Z 61.000,A 180.000,B 0.000,C 180.000} C_DIS
LIN {X 77.053,Y 10.040,Z 61.000,A 180.000,B 0.000,C 180.000} C_DIS
LIN {X 76.874,Y 10.080,Z 61.000,A 180.000,B 0.000,C 180.000} C_DIS
LIN {X 76.696,Y 10.133,Z 61.000,A 180.000,B 0.000,C 180.000} C_DIS
LIN {X 76.537,Y 10.193,Z 61.000,A 180.000,B 0.000,C 180.000} C_DIS
LIN {X 76.517,Y 10.201,Z 61.000,A 180.000,B 0.000,C 180.000} C_DIS
LIN {X 76.338,Y 10.286,Z 61.000,A 180.000,B 0.000,C 180.000} C_DIS
LIN {X 76.188,Y 10.372,Z 61.000,A 180.000,B 0.000,C 180.000} C_DIS
LIN {X 76.159,Y 10.390,Z 61.000,A 180.000,B 0.000,C 180.000} C_DIS
LIN {X 75.980,Y 10.515,Z 61.000,A 180.000,B 0.000,C 180.000} C_DIS
LIN {X 75.935,Y 10.551,Z 61.000,A 180.000,B 0.000,C 180.000} C_DIS
LIN {X 75.802,Y 10.665,Z 61.000,A 180.000,B 0.000,C 180.000} C_DIS
LIN {X 75.735,Y 10.729,Z 61.000,A 180.000,B 0.000,C 180.000} C_DIS
LIN {X 10.729,Y 75.735,Z 61.000,A 180.000,B 0.000,C 180.000} C_DIS
LIN {X 10.665,Y 75.802,Z 61.000,A 180.000,B 0.000,C 180.000} C_DIS
LIN {X 10.551,Y 75.935,Z 61.000,A 180.000,B 0.000,C 180.000} C_DIS
LIN {X 10.515,Y 75.980,Z 61.000,A 180.000,B 0.000,C 180.000} C_DIS
LIN {X 10.390,Y 76.159,Z 61.000,A 180.000,B 0.000,C 180.000} C_DIS
LIN {X 10.372,Y 76.188,Z 61.000,A 180.000,B 0.000,C 180.000} C_DIS
LIN {X 10.286,Y 76.338,Z 61.000,A 180.000,B 0.000,C 180.000} C_DIS
LIN {X 10.201,Y 76.517,Z 61.000,A 180.000,B 0.000,C 180.000} C_DIS
LIN {X 10.193,Y 76.537,Z 61.000,A 180.000,B 0.000,C 180.000} C_DIS
LIN {X 10.133,Y 76.696,Z 61.000,A 180.000,B 0.000,C 180.000} C_DIS
LIN {X 10.080,Y 76.874,Z 61.000,A 180.000,B 0.000,C 180.000} C_DIS
LIN {X 10.040,Y 77.053,Z 61.000,A 180.000,B 0.000,C 180.000} C_DIS
LIN {X 10.014,Y 77.232,Z 61.000,A 180.000,B 0.000,C 180.000} C_DIS
LIN {X 10.014,Y 77.233,Z 61.000,A 180.000,B 0.000,C 180.000} C_DIS
LIN {X 10.002,Y 77.411,Z 61.000,A 180.000,B 0.000,C 180.000} C_DIS
LIN {X 10.002,Y 77.589,Z 61.000,A 180.000,B 0.000,C 180.000} C_DIS
LIN {X 10.014,Y 77.767,Z 61.000,A 180.000,B 0.000,C 180.000} C_DIS
LIN {X 10.014,Y 77.768,Z 61.000,A 180.000,B 0.000,C 180.000} C_DIS
LIN {X 10.040,Y 77.947,Z 61.000,A 180.000,B 0.000,C 180.000} C_DIS
LIN {X 10.080,Y 78.126,Z 61.000,A 180.000,B 0.000,C 180.000} C_DIS
LIN {X 10.133,Y 78.304,Z 61.000,A 180.000,B 0.000,C 180.000} C_DIS
LIN {X 10.193,Y 78.463,Z 61.000,A 180.000,B 0.000,C 180.000} C_DIS
LIN {X 10.201,Y 78.483,Z 61.000,A 180.000,B 0.000,C 180.000} C_DIS
LIN {X 10.286,Y 78.662,Z 61.000,A 180.000,B 0.000,C 180.000} C_DIS
LIN {X 10.372,Y 78.812,Z 61.000,A 180.000,B 0.000,C 180.000} C_DIS
LIN {X 10.390,Y 78.841,Z 61.000,A 180.000,B 0.000,C 180.000} C_DIS
LIN {X 10.515,Y 79.020,Z 61.000,A 180.000,B 0.000,C 180.000} C_DIS
LIN {X 10.551,Y 79.065,Z 61.000,A 180.000,B 0.000,C 180.000} C_DIS
LIN {X 10.665,Y 79.198,Z 61.000,A 180.000,B 0.000,C 180.000} C_DIS
LIN {X 10.729,Y 79.265,Z 61.000,A 180.000,B 0.000,C 180.000} C_DIS
LIN {X 75.735,Y 144.271,Z 61.000,A 180.000,B 0.000,C 180.000} C_DIS
LIN {X 75.802,Y 144.335,Z 61.000,A 180.000,B 0.000,C 180.000} C_DIS
LIN {X 75.935,Y 144.449,Z 61.000,A 180.000,B 0.000,C 180.000} C_DIS
LIN {X 75.980,Y 144.485,Z 61.000,A 180.000,B 0.000,C 180.000} C_DIS
LIN {X 76.159,Y 144.610,Z 61.000,A 180.000,B 0.000,C 180.000} C_DIS
LIN {X 76.188,Y 144.628,Z 61.000,A 180.000,B 0.000,C 180.000} C_DIS
LIN {X 76.338,Y 144.714,Z 61.000,A 180.000,B 0.000,C 180.000} C_DIS
LIN {X 76.517,Y 144.799,Z 61.000,A 180.000,B 0.000,C 180.000} C_DIS
LIN {X 76.537,Y 144.807,Z 61.000,A 180.000,B 0.000,C 180.000} C_DIS
LIN {X 76.696,Y 144.867,Z 61.000,A 180.000,B 0.000,C 180.000} C_DIS
LIN {X 76.874,Y 144.920,Z 61.000,A 180.000,B 0.000,C 180.000} C_DIS
LIN {X 77.053,Y 144.960,Z 61.000,A 180.000,B 0.000,C 180.000} C_DIS
LIN {X 77.232,Y 144.986,Z 61.000,A 180.000,B 0.000,C 180.000} C_DIS
LIN {X 77.233,Y 144.986,Z 61.000,A 180.000,B 0.000,C 180.000} C_DIS
LIN {X 77.411,Y 144.998,Z 61.000,A 180.000,B 0.000,C 180.000} C_DIS
LIN {X 77.589,Y 144.998,Z 61.000,A 180.000,B 0.000,C 180.000} C_DIS
LIN {X 77.767,Y 144.986,Z 61.000,A 180.000,B 0.000,C 180.000} C_DIS
LIN {X 77.768,Y 144.986,Z 61.000,A 180.000,B 0.000,C 180.000} C_DIS
LIN {X 77.947,Y 144.960,Z 61.000,A 180.000,B 0.000,C 180.000} C_DIS
LIN {X 78.126,Y 144.920,Z 61.000,A 180.000,B 0.000,C 180.000} C_DIS
LIN {X 78.304,Y 144.867,Z 61.000,A 180.000,B 0.000,C 180.000} C_DIS
LIN {X 78.463,Y 144.807,Z 61.000,A 180.000,B 0.000,C 180.000} C_DIS
LIN {X 78.483,Y 144.799,Z 61.000,A 180.000,B 0.000,C 180.000} C_DIS
LIN {X 78.662,Y 144.714,Z 61.000,A 180.000,B 0.000,C 180.000} C_DIS
LIN {X 78.812,Y 144.628,Z 61.000,A 180.000,B 0.000,C 180.000} C_DIS
LIN {X 78.841,Y 144.610,Z 61.000,A 180.000,B 0.000,C 180.000} C_DIS
LIN {X 79.020,Y 144.485,Z 61.000,A 180.000,B 0.000,C 180.000} C_DIS
LIN {X 79.065,Y 144.449,Z 61.000,A 180.000,B 0.000,C 180.000} C_DIS
LIN {X 79.198,Y 144.335,Z 61.000,A 180.000,B 0.000,C 180.000} C_DIS
LIN {X 79.265,Y 144.271,Z 61.000,A 180.000,B 0.000,C 180.000} C_DIS
LIN {X 144.271,Y 79.265,Z 61.000,A 180.000,B 0.000,C 180.000} C_DIS
LIN {X 144.335,Y 79.198,Z 61.000,A 180.000,B 0.000,C 180.000} C_DIS
LIN {X 144.449,Y 79.065,Z 61.000,A 180.000,B 0.000,C 180.000} C_DIS
LIN {X 144.485,Y 79.020,Z 61.000,A 180.000,B 0.000,C 180.000} C_DIS
LIN {X 144.610,Y 78.841,Z 61.000,A 180.000,B 0.000,C 180.000} C_DIS
LIN {X 144.628,Y 78.812,Z 61.000,A 180.000,B 0.000,C 180.000} C_DIS
LIN {X 144.714,Y 78.662,Z 61.000,A 180.000,B 0.000,C 180.000} C_DIS
LIN {X 144.799,Y 78.483,Z 61.000,A 180.000,B 0.000,C 180.000} C_DIS
LIN {X 144.807,Y 78.463,Z 61.000,A 180.000,B 0.000,C 180.000} C_DIS
LIN {X 144.867,Y 78.304,Z 61.000,A 180.000,B 0.000,C 180.000} C_DIS
LIN {X 144.920,Y 78.126,Z 61.000,A 180.000,B 0.000,C 180.000} C_DIS
LIN {X 144.960,Y 77.947,Z 61.000,A 180.000,B 0.000,C 180.000} C_DIS
LIN {X 144.986,Y 77.768,Z 61.000,A 180.000,B 0.000,C 180.000} C_DIS
LIN {X 144.986,Y 77.767,Z 61.000,A 180.000,B 0.000,C 180.000} C_DIS
LIN {X 144.998,Y 77.589,Z 61.000,A 180.000,B 0.000,C 180.000} C_DIS
LIN {X 144.998,Y 77.411,Z 61.000,A 180.000,B 0.000,C 180.000} C_DIS
LIN {X 144.986,Y 77.233,Z 61.000,A 180.000,B 0.000,C 180.000} C_DIS
LIN {X 144.986,Y 77.232,Z 61.000,A 180.000,B 0.000,C 180.000} C_DIS
LIN {X 144.960,Y 77.053,Z 61.000,A 180.000,B 0.000,C 180.000} C_DIS
LIN {X 144.920,Y 76.874,Z 61.000,A 180.000,B 0.000,C 180.000} C_DIS
LIN {X 144.867,Y 76.696,Z 61.000,A 180.000,B 0.000,C 180.000} C_DIS
LIN {X 144.807,Y 76.537,Z 61.000,A 180.000,B 0.000,C 180.000} C_DIS
LIN {X 144.799,Y 76.517,Z 61.000,A 180.000,B 0.000,C 180.000} C_DIS
LIN {X 144.714,Y 76.338,Z 61.000,A 180.000,B 0.000,C 180.000} C_DIS
LIN {X 144.628,Y 76.188,Z 61.000,A 180.000,B 0.000,C 180.000} C_DIS
LIN {X 144.610,Y 76.159,Z 61.000,A 180.000,B 0.000,C 180.000} C_DIS
LIN {X 144.485,Y 75.980,Z 61.000,A 180.000,B 0.000,C 180.000} C_DIS
LIN {X 144.449,Y 75.935,Z 61.000,A 180.000,B 0.000,C 180.000} C_DIS
LIN {X 144.335,Y 75.802,Z 61.000,A 180.000,B 0.000,C 180.000} C_DIS
LIN {X 144.271,Y 75.735,Z 61.000,A 180.000,B 0.000,C 180.000} C_DIS
LIN {X 113.260,Y 44.725,Z 61.000,A 180.000,B 0.000,C 180.000} C_DIS
; Link Move Starts
LIN {X 113.037,Y 44.502,Z 61.000,A 180.000,B 0.000,C 180.000} C_DIS
LIN {X 112.815,Y 44.279,Z 60.999,A 180.000,B 0.000,C 180.000} C_DIS
LIN {X 112.592,Y 44.056,Z 60.998,A 180.000,B 0.000,C 180.000} C_DIS
LIN {X 112.369,Y 43.834,Z 60.996,A 180.000,B 0.000,C 180.000} C_DIS
LIN {X 112.147,Y 43.611,Z 60.994,A 180.000,B 0.000,C 180.000} C_DIS
LIN {X 111.924,Y 43.388,Z 60.991,A 180.000,B 0.000,C 180.000} C_DIS
LIN {X 111.701,Y 43.165,Z 60.988,A 180.000,B 0.000,C 180.000} C_DIS
LIN {X 111.478,Y 42.943,Z 60.985,A 180.000,B 0.000,C 180.000} C_DIS
LIN {X 111.256,Y 42.720,Z 60.981,A 180.000,B 0.000,C 180.000} C_DIS
LIN {X 111.033,Y 42.497,Z 60.977,A 180.000,B 0.000,C 180.000} C_DIS
LIN {X 110.810,Y 42.275,Z 60.972,A 180.000,B 0.000,C 180.000} C_DIS
LIN {X 110.699,Y 42.163,Z 60.969,A 180.000,B 0.000,C 180.000} C_DIS
LIN {X 110.587,Y 42.052,Z 60.967,A 180.000,B 0.000,C 180.000} C_DIS
LIN {X 110.476,Y 41.940,Z 60.964,A 180.000,B 0.000,C 180.000} C_DIS
LIN {X 110.365,Y 41.829,Z 60.961,A 180.000,B 0.000,C 180.000} C_DIS
LIN {X 110.253,Y 41.718,Z 60.959,A 180.000,B 0.000,C 180.000} C_DIS
LIN {X 110.142,Y 41.606,Z 60.956,A 180.000,B 0.000,C 180.000} C_DIS
LIN {X 110.030,Y 41.495,Z 60.952,A 180.000,B 0.000,C 180.000} C_DIS
LIN {X 109.919,Y 41.384,Z 60.949,A 180.000,B 0.000,C 180.000} C_DIS
LIN {X 109.808,Y 41.272,Z 60.946,A 180.000,B 0.000,C 180.000} C_DIS
LIN {X 109.696,Y 41.161,Z 60.943,A 180.000,B 0.000,C 180.000} C_DIS
LIN {X 109.585,Y 41.049,Z 60.939,A 180.000,B 0.000,C 180.000} C_DIS
LIN {X 109.474,Y 40.938,Z 60.936,A 180.000,B 0.000,C 180.000} C_DIS
LIN {X 109.362,Y 40.827,Z 60.932,A 180.000,B 0.000,C 180.000} C_DIS
LIN {X 109.251,Y 40.715,Z 60.928,A 180.000,B 0.000,C 180.000} C_DIS
LIN {X 109.140,Y 40.604,Z 60.925,A 180.000,B 0.000,C 180.000} C_DIS
LIN {X 109.028,Y 40.493,Z 60.921,A 180.000,B 0.000,C 180.000} C_DIS
LIN {X 108.917,Y 40.381,Z 60.917,A 180.000,B 0.000,C 180.000} C_DIS
LIN {X 108.805,Y 40.270,Z 60.913,A 180.000,B 0.000,C 180.000} C_DIS
LIN {X 108.694,Y 40.159,Z 60.909,A 180.000,B 0.000,C 180.000} C_DIS
LIN {X 108.583,Y 40.047,Z 60.905,A 180.000,B 0.000,C 180.000} C_DIS
LIN {X 108.471,Y 39.936,Z 60.900,A 180.000,B 0.000,C 180.000} C_DIS
LIN {X 108.360,Y 39.824,Z 60.896,A 180.000,B 0.000,C 180.000} C_DIS
LIN {X 108.249,Y 39.713,Z 60.892,A 180.000,B 0.000,C 180.000} C_DIS
LIN {X 108.137,Y 39.602,Z 60.887,A 180.000,B 0.000,C 180.000} C_DIS
LIN {X 108.026,Y 39.490,Z 60.883,A 180.000,B 0.000,C 180.000} C_DIS
LIN {X 107.914,Y 39.379,Z 60.878,A 180.000,B 0.000,C 180.000} C_DIS
LIN {X 107.803,Y 39.268,Z 60.873,A 180.000,B 0.000,C 180.000} C_DIS
LIN {X 107.692,Y 39.156,Z 60.869,A 180.000,B 0.000,C 180.000} C_DIS
LIN {X 107.580,Y 39.045,Z 60.864,A 180.000,B 0.000,C 180.000} C_DIS
LIN {X 107.469,Y 38.933,Z 60.859,A 180.000,B 0.000,C 180.000} C_DIS
LIN {X 107.358,Y 38.822,Z 60.854,A 180.000,B 0.000,C 180.000} C_DIS
LIN {X 107.302,Y 38.766,Z 60.851,A 180.000,B 0.000,C 180.000} C_DIS
LIN {X 107.246,Y 38.711,Z 60.849,A 180.000,B 0.000,C 180.000} C_DIS
LIN {X 107.191,Y 38.655,Z 60.846,A 180.000,B 0.000,C 180.000} C_DIS
LIN {X 107.135,Y 38.599,Z 60.844,A 180.000,B 0.000,C 180.000} C_DIS
LIN {X 107.079,Y 38.544,Z 60.841,A 180.000,B 0.000,C 180.000} C_DIS
LIN {X 107.024,Y 38.488,Z 60.839,A 180.000,B 0.000,C 180.000} C_DIS
LIN {X 106.968,Y 38.432,Z 60.836,A 180.000,B 0.000,C 180.000} C_DIS
LIN {X 106.856,Y 38.321,Z 60.831,A 180.000,B 0.000,C 180.000} C_DIS
LIN {X 106.745,Y 38.210,Z 60.825,A 180.000,B 0.000,C 180.000} C_DIS
LIN {X 106.634,Y 38.098,Z 60.820,A 180.000,B 0.000,C 180.000} C_DIS
LIN {X 106.522,Y 37.987,Z 60.815,A 180.000,B 0.000,C 180.000} C_DIS
LIN {X 106.411,Y 37.875,Z 60.809,A 180.000,B 0.000,C 180.000} C_DIS
LIN {X 106.355,Y 37.820,Z 60.806,A 180.000,B 0.000,C 180.000} C_DIS
LIN {X 106.244,Y 37.708,Z 60.801,A 180.000,B 0.000,C 180.000} C_DIS
LIN {X 106.077,Y 37.541,Z 60.793,A 180.000,B 0.000,C 180.000} C_DIS
LIN {X 105.966,Y 37.430,Z 60.787,A 180.000,B 0.000,C 180.000} C_DIS
LIN {X 105.910,Y 37.374,Z 60.785,A 180.000,B 0.000,C 180.000} C_DIS
LIN {X 105.798,Y 37.263,Z 60.779,A 180.000,B 0.000,C 180.000} C_DIS
LIN {X 105.631,Y 37.096,Z 60.771,A 180.000,B 0.000,C 180.000} C_DIS
LIN {X 105.520,Y 36.985,Z 60.765,A 180.000,B 0.000,C 180.000} C_DIS
LIN {X 105.464,Y 36.929,Z 60.763,A 180.000,B 0.000,C 180.000} C_DIS
LIN {X 105.353,Y 36.817,Z 60.757,A 180.000,B 0.000,C 180.000} C_DIS
LIN {X 105.186,Y 36.650,Z 60.749,A 180.000,B 0.000,C 180.000} C_DIS
LIN {X 105.075,Y 36.539,Z 60.743,A 180.000,B 0.000,C 180.000} C_DIS
LIN {X 105.019,Y 36.483,Z 60.741,A 180.000,B 0.000,C 180.000} C_DIS
LIN {X 104.908,Y 36.372,Z 60.735,A 180.000,B 0.000,C 180.000} C_DIS
LIN {X 104.740,Y 36.205,Z 60.727,A 180.000,B 0.000,C 180.000} C_DIS
LIN {X 104.629,Y 36.094,Z 60.721,A 180.000,B 0.000,C 180.000} C_DIS
LIN {X 104.573,Y 36.038,Z 60.719,A 180.000,B 0.000,C 180.000} C_DIS
LIN {X 104.462,Y 35.927,Z 60.713,A 180.000,B 0.000,C 180.000} C_DIS
LIN {X 104.128,Y 35.592,Z 60.697,A 180.000,B 0.000,C 180.000} C_DIS
LIN {X 104.017,Y 35.481,Z 60.691,A 180.000,B 0.000,C 180.000} C_DIS
LIN {X 103.682,Y 35.147,Z 60.675,A 180.000,B 0.000,C 180.000} C_DIS
LIN {X 103.571,Y 35.036,Z 60.669,A 180.000,B 0.000,C 180.000} C_DIS
LIN {X 103.181,Y 34.646,Z 60.650,A 180.000,B 0.000,C 180.000} C_DIS
LIN {X 102.847,Y 34.312,Z 60.633,A 180.000,B 0.000,C 180.000} C_DIS
LIN {X 102.736,Y 34.200,Z 60.628,A 180.000,B 0.000,C 180.000} C_DIS
LIN {X 102.402,Y 33.866,Z 60.611,A 180.000,B 0.000,C 180.000} C_DIS
LIN {X 102.290,Y 33.755,Z 60.606,A 180.000,B 0.000,C 180.000} C_DIS
LIN {X 101.734,Y 33.198,Z 60.578,A 180.000,B 0.000,C 180.000} C_DIS
LIN {X 101.455,Y 32.920,Z 60.565,A 180.000,B 0.000,C 180.000} C_DIS
LIN {X 101.121,Y 32.585,Z 60.548,A 180.000,B 0.000,C 180.000} C_DIS
LIN {X 99.840,Y 31.305,Z 60.485,A 180.000,B 0.000,C 180.000} C_DIS
LIN {X 97.724,Y 29.189,Z 60.380,A 180.000,B 0.000,C 180.000} C_DIS
LIN {X 97.613,Y 29.077,Z 60.375,A 180.000,B 0.000,C 180.000} C_DIS
LIN {X 97.279,Y 28.743,Z 60.358,A 180.000,B 0.000,C 180.000} C_DIS
LIN {X 97.167,Y 28.632,Z 60.353,A 180.000,B 0.000,C 180.000} C_DIS
LIN {X 96.833,Y 28.298,Z 60.336,A 180.000,B 0.000,C 180.000} C_DIS
LIN {X 96.778,Y 28.242,Z 60.334,A 180.000,B 0.000,C 180.000} C_DIS
LIN {X 96.666,Y 28.131,Z 60.328,A 180.000,B 0.000,C 180.000} C_DIS
LIN {X 96.332,Y 27.797,Z 60.312,A 180.000,B 0.000,C 180.000} C_DIS
LIN {X 96.221,Y 27.685,Z 60.306,A 180.000,B 0.000,C 180.000} C_DIS
LIN {X 95.887,Y 27.351,Z 60.290,A 180.000,B 0.000,C 180.000} C_DIS
LIN {X 95.775,Y 27.240,Z 60.284,A 180.000,B 0.000,C 180.000} C_DIS
LIN {X 95.608,Y 27.073,Z 60.276,A 180.000,B 0.000,C 180.000} C_DIS
LIN {X 95.497,Y 26.961,Z 60.270,A 180.000,B 0.000,C 180.000} C_DIS
LIN {X 95.441,Y 26.906,Z 60.268,A 180.000,B 0.000,C 180.000} C_DIS
LIN {X 95.330,Y 26.794,Z 60.262,A 180.000,B 0.000,C 180.000} C_DIS
LIN {X 95.163,Y 26.627,Z 60.254,A 180.000,B 0.000,C 180.000} C_DIS
LIN {X 95.051,Y 26.516,Z 60.248,A 180.000,B 0.000,C 180.000} C_DIS
LIN {X 94.996,Y 26.460,Z 60.246,A 180.000,B 0.000,C 180.000} C_DIS
LIN {X 94.884,Y 26.349,Z 60.240,A 180.000,B 0.000,C 180.000} C_DIS
LIN {X 94.717,Y 26.182,Z 60.232,A 180.000,B 0.000,C 180.000} C_DIS
LIN {X 94.606,Y 26.070,Z 60.226,A 180.000,B 0.000,C 180.000} C_DIS
LIN {X 94.550,Y 26.015,Z 60.224,A 180.000,B 0.000,C 180.000} C_DIS
LIN {X 94.439,Y 25.903,Z 60.218,A 180.000,B 0.000,C 180.000} C_DIS
LIN {X 94.272,Y 25.736,Z 60.210,A 180.000,B 0.000,C 180.000} C_DIS
LIN {X 94.160,Y 25.625,Z 60.204,A 180.000,B 0.000,C 180.000} C_DIS
LIN {X 94.105,Y 25.569,Z 60.202,A 180.000,B 0.000,C 180.000} C_DIS
LIN {X 93.993,Y 25.458,Z 60.196,A 180.000,B 0.000,C 180.000} C_DIS
LIN {X 93.882,Y 25.346,Z 60.191,A 180.000,B 0.000,C 180.000} C_DIS
LIN {X 93.771,Y 25.235,Z 60.185,A 180.000,B 0.000,C 180.000} C_DIS
LIN {X 93.659,Y 25.124,Z 60.180,A 180.000,B 0.000,C 180.000} C_DIS
LIN {X 93.548,Y 25.012,Z 60.174,A 180.000,B 0.000,C 180.000} C_DIS
LIN {X 93.437,Y 24.901,Z 60.169,A 180.000,B 0.000,C 180.000} C_DIS
LIN {X 93.325,Y 24.790,Z 60.164,A 180.000,B 0.000,C 180.000} C_DIS
LIN {X 93.269,Y 24.734,Z 60.161,A 180.000,B 0.000,C 180.000} C_DIS
LIN {X 93.214,Y 24.678,Z 60.159,A 180.000,B 0.000,C 180.000} C_DIS
LIN {X 93.158,Y 24.623,Z 60.156,A 180.000,B 0.000,C 180.000} C_DIS
LIN {X 93.102,Y 24.567,Z 60.154,A 180.000,B 0.000,C 180.000} C_DIS
LIN {X 93.047,Y 24.511,Z 60.151,A 180.000,B 0.000,C 180.000} C_DIS
LIN {X 92.991,Y 24.456,Z 60.148,A 180.000,B 0.000,C 180.000} C_DIS
LIN {X 92.880,Y 24.344,Z 60.143,A 180.000,B 0.000,C 180.000} C_DIS
LIN {X 92.768,Y 24.233,Z 60.139,A 180.000,B 0.000,C 180.000} C_DIS
LIN {X 92.657,Y 24.121,Z 60.134,A 180.000,B 0.000,C 180.000} C_DIS
LIN {X 92.546,Y 24.010,Z 60.129,A 180.000,B 0.000,C 180.000} C_DIS
LIN {X 92.434,Y 23.899,Z 60.124,A 180.000,B 0.000,C 180.000} C_DIS
LIN {X 92.323,Y 23.787,Z 60.120,A 180.000,B 0.000,C 180.000} C_DIS
LIN {X 92.211,Y 23.676,Z 60.115,A 180.000,B 0.000,C 180.000} C_DIS
LIN {X 92.100,Y 23.565,Z 60.110,A 180.000,B 0.000,C 180.000} C_DIS
LIN {X 91.989,Y 23.453,Z 60.106,A 180.000,B 0.000,C 180.000} C_DIS
LIN {X 91.877,Y 23.342,Z 60.102,A 180.000,B 0.000,C 180.000} C_DIS
LIN {X 91.766,Y 23.230,Z 60.097,A 180.000,B 0.000,C 180.000} C_DIS
LIN {X 91.655,Y 23.119,Z 60.093,A 180.000,B 0.000,C 180.000} C_DIS
LIN {X 91.543,Y 23.008,Z 60.089,A 180.000,B 0.000,C 180.000} C_DIS
LIN {X 91.432,Y 22.896,Z 60.085,A 180.000,B 0.000,C 180.000} C_DIS
LIN {X 91.321,Y 22.785,Z 60.081,A 180.000,B 0.000,C 180.000} C_DIS
LIN {X 91.209,Y 22.674,Z 60.077,A 180.000,B 0.000,C 180.000} C_DIS
LIN {X 91.098,Y 22.562,Z 60.073,A 180.000,B 0.000,C 180.000} C_DIS
LIN {X 90.986,Y 22.451,Z 60.070,A 180.000,B 0.000,C 180.000} C_DIS
LIN {X 90.875,Y 22.340,Z 60.066,A 180.000,B 0.000,C 180.000} C_DIS
LIN {X 90.764,Y 22.228,Z 60.062,A 180.000,B 0.000,C 180.000} C_DIS
LIN {X 90.652,Y 22.117,Z 60.059,A 180.000,B 0.000,C 180.000} C_DIS
LIN {X 90.541,Y 22.005,Z 60.056,A 180.000,B 0.000,C 180.000} C_DIS
LIN {X 90.430,Y 21.894,Z 60.052,A 180.000,B 0.000,C 180.000} C_DIS
LIN {X 90.318,Y 21.783,Z 60.049,A 180.000,B 0.000,C 180.000} C_DIS
LIN {X 90.207,Y 21.671,Z 60.046,A 180.000,B 0.000,C 180.000} C_DIS
LIN {X 90.095,Y 21.560,Z 60.043,A 180.000,B 0.000,C 180.000} C_DIS
LIN {X 89.984,Y 21.449,Z 60.040,A 180.000,B 0.000,C 180.000} C_DIS
LIN {X 89.873,Y 21.337,Z 60.037,A 180.000,B 0.000,C 180.000} C_DIS
LIN {X 89.761,Y 21.226,Z 60.034,A 180.000,B 0.000,C 180.000} C_DIS
LIN {X 89.650,Y 21.114,Z 60.032,A 180.000,B 0.000,C 180.000} C_DIS
LIN {X 89.539,Y 21.003,Z 60.029,A 180.000,B 0.000,C 180.000} C_DIS
LIN {X 89.427,Y 20.892,Z 60.027,A 180.000,B 0.000,C 180.000} C_DIS
LIN {X 89.205,Y 20.669,Z 60.022,A 180.000,B 0.000,C 180.000} C_DIS
LIN {X 88.982,Y 20.446,Z 60.018,A 180.000,B 0.000,C 180.000} C_DIS
LIN {X 88.759,Y 20.224,Z 60.014,A 180.000,B 0.000,C 180.000} C_DIS
LIN {X 88.536,Y 20.001,Z 60.011,A 180.000,B 0.000,C 180.000} C_DIS
LIN {X 88.314,Y 19.778,Z 60.008,A 180.000,B 0.000,C 180.000} C_DIS
LIN {X 88.091,Y 19.555,Z 60.005,A 180.000,B 0.000,C 180.000} C_DIS
LIN {X 87.868,Y 19.333,Z 60.003,A 180.000,B 0.000,C 180.000} C_DIS
LIN {X 87.645,Y 19.110,Z 60.002,A 180.000,B 0.000,C 180.000} C_DIS
LIN {X 87.423,Y 18.887,Z 60.001,A 180.000,B 0.000,C 180.000} C_DIS
LIN {X 87.200,Y 18.664,Z 60.000,A 180.000,B 0.000,C 180.000} C_DIS
LIN {X 87.037,Y 18.501,Z 60.000,A 180.000,B 0.000,C 180.000} C_DIS
; Cutting Move Starts
LIN {X 79.265,Y 10.729,Z 60.000,A 180.000,B 0.000,C 180.000} C_DIS
LIN {X 79.198,Y 10.665,Z 60.000,A 180.000,B 0.000,C 180.000} C_DIS
LIN {X 79.065,Y 10.551,Z 60.000,A 180.000,B 0.000,C 180.000} C_DIS
LIN {X 79.020,Y 10.515,Z 60.000,A 180.000,B 0.000,C 180.000} C_DIS
LIN {X 78.841,Y 10.390,Z 60.000,A 180.000,B 0.000,C 180.000} C_DIS
LIN {X 78.812,Y 10.372,Z 60.000,A 180.000,B 0.000,C 180.000} C_DIS
LIN {X 78.662,Y 10.286,Z 60.000,A 180.000,B 0.000,C 180.000} C_DIS
LIN {X 78.483,Y 10.201,Z 60.000,A 180.000,B 0.000,C 180.000} C_DIS
LIN {X 78.463,Y 10.193,Z 60.000,A 180.000,B 0.000,C 180.000} C_DIS
LIN {X 78.304,Y 10.133,Z 60.000,A 180.000,B 0.000,C 180.000} C_DIS
LIN {X 78.126,Y 10.080,Z 60.000,A 180.000,B 0.000,C 180.000} C_DIS
LIN {X 77.947,Y 10.040,Z 60.000,A 180.000,B 0.000,C 180.000} C_DIS
LIN {X 77.768,Y 10.014,Z 60.000,A 180.000,B 0.000,C 180.000} C_DIS
LIN {X 77.767,Y 10.014,Z 60.000,A 180.000,B 0.000,C 180.000} C_DIS
LIN {X 77.589,Y 10.002,Z 60.000,A 180.000,B 0.000,C 180.000} C_DIS
LIN {X 77.411,Y 10.002,Z 60.000,A 180.000,B 0.000,C 180.000} C_DIS
LIN {X 77.233,Y 10.014,Z 60.000,A 180.000,B 0.000,C 180.000} C_DIS
LIN {X 77.232,Y 10.014,Z 60.000,A 180.000,B 0.000,C 180.000} C_DIS
LIN {X 77.053,Y 10.040,Z 60.000,A 180.000,B 0.000,C 180.000} C_DIS
LIN {X 76.874,Y 10.080,Z 60.000,A 180.000,B 0.000,C 180.000} C_DIS
LIN {X 76.696,Y 10.133,Z 60.000,A 180.000,B 0.000,C 180.000} C_DIS
LIN {X 76.537,Y 10.193,Z 60.000,A 180.000,B 0.000,C 180.000} C_DIS
LIN {X 76.517,Y 10.201,Z 60.000,A 180.000,B 0.000,C 180.000} C_DIS
LIN {X 76.338,Y 10.286,Z 60.000,A 180.000,B 0.000,C 180.000} C_DIS
LIN {X 76.188,Y 10.372,Z 60.000,A 180.000,B 0.000,C 180.000} C_DIS
LIN {X 76.159,Y 10.390,Z 60.000,A 180.000,B 0.000,C 180.000} C_DIS
LIN {X 75.980,Y 10.515,Z 60.000,A 180.000,B 0.000,C 180.000} C_DIS
LIN {X 75.935,Y 10.551,Z 60.000,A 180.000,B 0.000,C 180.000} C_DIS
LIN {X 75.802,Y 10.665,Z 60.000,A 180.000,B 0.000,C 180.000} C_DIS
LIN {X 75.735,Y 10.729,Z 60.000,A 180.000,B 0.000,C 180.000} C_DIS
LIN {X 10.729,Y 75.735,Z 60.000,A 180.000,B 0.000,C 180.000} C_DIS
LIN {X 10.665,Y 75.802,Z 60.000,A 180.000,B 0.000,C 180.000} C_DIS
LIN {X 10.551,Y 75.935,Z 60.000,A 180.000,B 0.000,C 180.000} C_DIS
LIN {X 10.515,Y 75.980,Z 60.000,A 180.000,B 0.000,C 180.000} C_DIS
LIN {X 10.390,Y 76.159,Z 60.000,A 180.000,B 0.000,C 180.000} C_DIS
LIN {X 10.372,Y 76.188,Z 60.000,A 180.000,B 0.000,C 180.000} C_DIS
LIN {X 10.286,Y 76.338,Z 60.000,A 180.000,B 0.000,C 180.000} C_DIS
LIN {X 10.201,Y 76.517,Z 60.000,A 180.000,B 0.000,C 180.000} C_DIS
LIN {X 10.193,Y 76.537,Z 60.000,A 180.000,B 0.000,C 180.000} C_DIS
LIN {X 10.133,Y 76.696,Z 60.000,A 180.000,B 0.000,C 180.000} C_DIS
LIN {X 10.080,Y 76.874,Z 60.000,A 180.000,B 0.000,C 180.000} C_DIS
LIN {X 10.040,Y 77.053,Z 60.000,A 180.000,B 0.000,C 180.000} C_DIS
LIN {X 10.014,Y 77.232,Z 60.000,A 180.000,B 0.000,C 180.000} C_DIS
LIN {X 10.014,Y 77.233,Z 60.000,A 180.000,B 0.000,C 180.000} C_DIS
LIN {X 10.002,Y 77.411,Z 60.000,A 180.000,B 0.000,C 180.000} C_DIS
LIN {X 10.002,Y 77.589,Z 60.000,A 180.000,B 0.000,C 180.000} C_DIS
LIN {X 10.014,Y 77.767,Z 60.000,A 180.000,B 0.000,C 180.000} C_DIS
LIN {X 10.014,Y 77.768,Z 60.000,A 180.000,B 0.000,C 180.000} C_DIS
LIN {X 10.040,Y 77.947,Z 60.000,A 180.000,B 0.000,C 180.000} C_DIS
LIN {X 10.080,Y 78.126,Z 60.000,A 180.000,B 0.000,C 180.000} C_DIS
LIN {X 10.133,Y 78.304,Z 60.000,A 180.000,B 0.000,C 180.000} C_DIS
LIN {X 10.193,Y 78.463,Z 60.000,A 180.000,B 0.000,C 180.000} C_DIS
LIN {X 10.201,Y 78.483,Z 60.000,A 180.000,B 0.000,C 180.000} C_DIS
LIN {X 10.286,Y 78.662,Z 60.000,A 180.000,B 0.000,C 180.000} C_DIS
LIN {X 10.372,Y 78.812,Z 60.000,A 180.000,B 0.000,C 180.000} C_DIS
LIN {X 10.390,Y 78.841,Z 60.000,A 180.000,B 0.000,C 180.000} C_DIS
LIN {X 10.515,Y 79.020,Z 60.000,A 180.000,B 0.000,C 180.000} C_DIS
LIN {X 10.551,Y 79.065,Z 60.000,A 180.000,B 0.000,C 180.000} C_DIS
LIN {X 10.665,Y 79.198,Z 60.000,A 180.000,B 0.000,C 180.000} C_DIS
LIN {X 10.729,Y 79.265,Z 60.000,A 180.000,B 0.000,C 180.000} C_DIS
LIN {X 75.735,Y 144.271,Z 60.000,A 180.000,B 0.000,C 180.000} C_DIS
LIN {X 75.802,Y 144.335,Z 60.000,A 180.000,B 0.000,C 180.000} C_DIS
LIN {X 75.935,Y 144.449,Z 60.000,A 180.000,B 0.000,C 180.000} C_DIS
LIN {X 75.980,Y 144.485,Z 60.000,A 180.000,B 0.000,C 180.000} C_DIS
LIN {X 76.159,Y 144.610,Z 60.000,A 180.000,B 0.000,C 180.000} C_DIS
LIN {X 76.188,Y 144.628,Z 60.000,A 180.000,B 0.000,C 180.000} C_DIS
LIN {X 76.338,Y 144.714,Z 60.000,A 180.000,B 0.000,C 180.000} C_DIS
LIN {X 76.517,Y 144.799,Z 60.000,A 180.000,B 0.000,C 180.000} C_DIS
LIN {X 76.537,Y 144.807,Z 60.000,A 180.000,B 0.000,C 180.000} C_DIS
LIN {X 76.696,Y 144.867,Z 60.000,A 180.000,B 0.000,C 180.000} C_DIS
LIN {X 76.874,Y 144.920,Z 60.000,A 180.000,B 0.000,C 180.000} C_DIS
LIN {X 77.053,Y 144.960,Z 60.000,A 180.000,B 0.000,C 180.000} C_DIS
LIN {X 77.232,Y 144.986,Z 60.000,A 180.000,B 0.000,C 180.000} C_DIS
LIN {X 77.233,Y 144.986,Z 60.000,A 180.000,B 0.000,C 180.000} C_DIS
LIN {X 77.411,Y 144.998,Z 60.000,A 180.000,B 0.000,C 180.000} C_DIS
LIN {X 77.589,Y 144.998,Z 60.000,A 180.000,B 0.000,C 180.000} C_DIS
LIN {X 77.767,Y 144.986,Z 60.000,A 180.000,B 0.000,C 180.000} C_DIS
LIN {X 77.768,Y 144.986,Z 60.000,A 180.000,B 0.000,C 180.000} C_DIS
LIN {X 77.947,Y 144.960,Z 60.000,A 180.000,B 0.000,C 180.000} C_DIS
LIN {X 78.126,Y 144.920,Z 60.000,A 180.000,B 0.000,C 180.000} C_DIS
LIN {X 78.304,Y 144.867,Z 60.000,A 180.000,B 0.000,C 180.000} C_DIS
LIN {X 78.463,Y 144.807,Z 60.000,A 180.000,B 0.000,C 180.000} C_DIS
LIN {X 78.483,Y 144.799,Z 60.000,A 180.000,B 0.000,C 180.000} C_DIS
LIN {X 78.662,Y 144.714,Z 60.000,A 180.000,B 0.000,C 180.000} C_DIS
LIN {X 78.812,Y 144.628,Z 60.000,A 180.000,B 0.000,C 180.000} C_DIS
LIN {X 78.841,Y 144.610,Z 60.000,A 180.000,B 0.000,C 180.000} C_DIS
LIN {X 79.020,Y 144.485,Z 60.000,A 180.000,B 0.000,C 180.000} C_DIS
LIN {X 79.065,Y 144.449,Z 60.000,A 180.000,B 0.000,C 180.000} C_DIS
LIN {X 79.198,Y 144.335,Z 60.000,A 180.000,B 0.000,C 180.000} C_DIS
LIN {X 79.265,Y 144.271,Z 60.000,A 180.000,B 0.000,C 180.000} C_DIS
LIN {X 144.271,Y 79.265,Z 60.000,A 180.000,B 0.000,C 180.000} C_DIS
LIN {X 144.335,Y 79.198,Z 60.000,A 180.000,B 0.000,C 180.000} C_DIS
LIN {X 144.449,Y 79.065,Z 60.000,A 180.000,B 0.000,C 180.000} C_DIS
LIN {X 144.485,Y 79.020,Z 60.000,A 180.000,B 0.000,C 180.000} C_DIS
LIN {X 144.610,Y 78.841,Z 60.000,A 180.000,B 0.000,C 180.000} C_DIS
LIN {X 144.628,Y 78.812,Z 60.000,A 180.000,B 0.000,C 180.000} C_DIS
LIN {X 144.714,Y 78.662,Z 60.000,A 180.000,B 0.000,C 180.000} C_DIS
LIN {X 144.799,Y 78.483,Z 60.000,A 180.000,B 0.000,C 180.000} C_DIS
LIN {X 144.807,Y 78.463,Z 60.000,A 180.000,B 0.000,C 180.000} C_DIS
LIN {X 144.867,Y 78.304,Z 60.000,A 180.000,B 0.000,C 180.000} C_DIS
LIN {X 144.920,Y 78.126,Z 60.000,A 180.000,B 0.000,C 180.000} C_DIS
LIN {X 144.960,Y 77.947,Z 60.000,A 180.000,B 0.000,C 180.000} C_DIS
LIN {X 144.986,Y 77.768,Z 60.000,A 180.000,B 0.000,C 180.000} C_DIS
LIN {X 144.986,Y 77.767,Z 60.000,A 180.000,B 0.000,C 180.000} C_DIS
LIN {X 144.998,Y 77.589,Z 60.000,A 180.000,B 0.000,C 180.000} C_DIS
LIN {X 144.998,Y 77.411,Z 60.000,A 180.000,B 0.000,C 180.000} C_DIS
LIN {X 144.986,Y 77.233,Z 60.000,A 180.000,B 0.000,C 180.000} C_DIS
LIN {X 144.986,Y 77.232,Z 60.000,A 180.000,B 0.000,C 180.000} C_DIS
LIN {X 144.960,Y 77.053,Z 60.000,A 180.000,B 0.000,C 180.000} C_DIS
LIN {X 144.920,Y 76.874,Z 60.000,A 180.000,B 0.000,C 180.000} C_DIS
LIN {X 144.867,Y 76.696,Z 60.000,A 180.000,B 0.000,C 180.000} C_DIS
LIN {X 144.807,Y 76.537,Z 60.000,A 180.000,B 0.000,C 180.000} C_DIS
LIN {X 144.799,Y 76.517,Z 60.000,A 180.000,B 0.000,C 180.000} C_DIS
LIN {X 144.714,Y 76.338,Z 60.000,A 180.000,B 0.000,C 180.000} C_DIS
LIN {X 144.628,Y 76.188,Z 60.000,A 180.000,B 0.000,C 180.000} C_DIS
LIN {X 144.610,Y 76.159,Z 60.000,A 180.000,B 0.000,C 180.000} C_DIS
LIN {X 144.485,Y 75.980,Z 60.000,A 180.000,B 0.000,C 180.000} C_DIS
LIN {X 144.449,Y 75.935,Z 60.000,A 180.000,B 0.000,C 180.000} C_DIS
LIN {X 144.335,Y 75.802,Z 60.000,A 180.000,B 0.000,C 180.000} C_DIS
LIN {X 144.271,Y 75.735,Z 60.000,A 180.000,B 0.000,C 180.000} C_DIS
LIN {X 113.260,Y 44.725,Z 60.000,A 180.000,B 0.000,C 180.000} C_DIS
LIN {X 87.037,Y 18.501,Z 60.000,A 180.000,B 0.000,C 180.000} C_DIS
; Link Move Starts
LIN {X 86.814,Y 18.278,Z 60.000,A 180.000,B 0.000,C 180.000} C_DIS
LIN {X 86.591,Y 18.056,Z 59.999,A 180.000,B 0.000,C 180.000} C_DIS
LIN {X 86.368,Y 17.833,Z 59.998,A 180.000,B 0.000,C 180.000} C_DIS
LIN {X 86.146,Y 17.610,Z 59.996,A 180.000,B 0.000,C 180.000} C_DIS
LIN {X 85.923,Y 17.387,Z 59.994,A 180.000,B 0.000,C 180.000} C_DIS
LIN {X 85.700,Y 17.165,Z 59.991,A 180.000,B 0.000,C 180.000} C_DIS
LIN {X 85.477,Y 16.942,Z 59.988,A 180.000,B 0.000,C 180.000} C_DIS
LIN {X 85.255,Y 16.719,Z 59.985,A 180.000,B 0.000,C 180.000} C_DIS
LIN {X 85.032,Y 16.496,Z 59.981,A 180.000,B 0.000,C 180.000} C_DIS
LIN {X 84.809,Y 16.274,Z 59.977,A 180.000,B 0.000,C 180.000} C_DIS
LIN {X 84.587,Y 16.051,Z 59.972,A 180.000,B 0.000,C 180.000} C_DIS
LIN {X 84.475,Y 15.940,Z 59.969,A 180.000,B 0.000,C 180.000} C_DIS
LIN {X 84.364,Y 15.828,Z 59.967,A 180.000,B 0.000,C 180.000} C_DIS
LIN {X 84.252,Y 15.717,Z 59.964,A 180.000,B 0.000,C 180.000} C_DIS
LIN {X 84.141,Y 15.605,Z 59.961,A 180.000,B 0.000,C 180.000} C_DIS
LIN {X 84.030,Y 15.494,Z 59.959,A 180.000,B 0.000,C 180.000} C_DIS
LIN {X 83.918,Y 15.383,Z 59.956,A 180.000,B 0.000,C 180.000} C_DIS
LIN {X 83.807,Y 15.271,Z 59.952,A 180.000,B 0.000,C 180.000} C_DIS
LIN {X 83.696,Y 15.160,Z 59.949,A 180.000,B 0.000,C 180.000} C_DIS
LIN {X 83.584,Y 15.049,Z 59.946,A 180.000,B 0.000,C 180.000} C_DIS
LIN {X 83.473,Y 14.937,Z 59.943,A 180.000,B 0.000,C 180.000} C_DIS
LIN {X 83.361,Y 14.826,Z 59.939,A 180.000,B 0.000,C 180.000} C_DIS
LIN {X 83.250,Y 14.715,Z 59.936,A 180.000,B 0.000,C 180.000} C_DIS
LIN {X 83.139,Y 14.603,Z 59.932,A 180.000,B 0.000,C 180.000} C_DIS
LIN {X 83.027,Y 14.492,Z 59.928,A 180.000,B 0.000,C 180.000} C_DIS
LIN {X 82.916,Y 14.380,Z 59.925,A 180.000,B 0.000,C 180.000} C_DIS
LIN {X 82.805,Y 14.269,Z 59.921,A 180.000,B 0.000,C 180.000} C_DIS
LIN {X 82.693,Y 14.158,Z 59.917,A 180.000,B 0.000,C 180.000} C_DIS
LIN {X 82.582,Y 14.046,Z 59.913,A 180.000,B 0.000,C 180.000} C_DIS
LIN {X 82.470,Y 13.935,Z 59.909,A 180.000,B 0.000,C 180.000} C_DIS
LIN {X 82.359,Y 13.824,Z 59.905,A 180.000,B 0.000,C 180.000} C_DIS
LIN {X 82.248,Y 13.712,Z 59.900,A 180.000,B 0.000,C 180.000} C_DIS
LIN {X 82.136,Y 13.601,Z 59.896,A 180.000,B 0.000,C 180.000} C_DIS
LIN {X 82.025,Y 13.489,Z 59.892,A 180.000,B 0.000,C 180.000} C_DIS
LIN {X 81.914,Y 13.378,Z 59.887,A 180.000,B 0.000,C 180.000} C_DIS
LIN {X 81.802,Y 13.267,Z 59.883,A 180.000,B 0.000,C 180.000} C_DIS
LIN {X 81.691,Y 13.155,Z 59.878,A 180.000,B 0.000,C 180.000} C_DIS
LIN {X 81.580,Y 13.044,Z 59.873,A 180.000,B 0.000,C 180.000} C_DIS
LIN {X 81.468,Y 12.933,Z 59.869,A 180.000,B 0.000,C 180.000} C_DIS
LIN {X 81.357,Y 12.821,Z 59.864,A 180.000,B 0.000,C 180.000} C_DIS
LIN {X 81.245,Y 12.710,Z 59.859,A 180.000,B 0.000,C 180.000} C_DIS
LIN {X 81.134,Y 12.599,Z 59.854,A 180.000,B 0.000,C 180.000} C_DIS
LIN {X 81.078,Y 12.543,Z 59.851,A 180.000,B 0.000,C 180.000} C_DIS
LIN {X 81.023,Y 12.487,Z 59.849,A 180.000,B 0.000,C 180.000} C_DIS
LIN {X 80.967,Y 12.431,Z 59.846,A 180.000,B 0.000,C 180.000} C_DIS
LIN {X 80.911,Y 12.376,Z 59.844,A 180.000,B 0.000,C 180.000} C_DIS
LIN {X 80.856,Y 12.320,Z 59.841,A 180.000,B 0.000,C 180.000} C_DIS
LIN {X 80.800,Y 12.264,Z 59.839,A 180.000,B 0.000,C 180.000} C_DIS
LIN {X 80.744,Y 12.209,Z 59.836,A 180.000,B 0.000,C 180.000} C_DIS
LIN {X 80.633,Y 12.097,Z 59.831,A 180.000,B 0.000,C 180.000} C_DIS
LIN {X 80.522,Y 11.986,Z 59.825,A 180.000,B 0.000,C 180.000} C_DIS
LIN {X 80.410,Y 11.875,Z 59.820,A 180.000,B 0.000,C 180.000} C_DIS
